(* IEC 61131-3 sources: Bachelor/LARS redcrane-simulation/plc_export/FB_InverceKinematics, 1 file *)

(* ---- RedCrane_kinematic_model.st ---- *)
(*
 *
 * File: RedCrane_kinematic_model.st
 *
 * IEC 61131-3 Structured Text (ST) code generated for subsystem "RedCrane_kinematic_model/FB_InverceKinematics"
 *
 * Model name                      : RedCrane_kinematic_model
 * Model version                   : 2.78
 * Model creator                   : sindr
 * Model last modified by          : larso
 * Model last modified on          : Mon Jan 20 08:44:51 2025
 * Model sample time               : 0.001s
 * Subsystem name                  : RedCrane_kinematic_model/FB_InverceKinematics
 * Subsystem sample time           : 0.001s
 * Simulink PLC Coder version      : 24.1 (R2024a) 19-Nov-2023
 * ST code generated on            : Mon Jan 20 09:25:34 2025
 *
 * Target IDE selection            : Beckhoff TwinCAT 3
 * Test Bench included             : No
 *
 *)
FUNCTION_BLOCK FB_InverceKinematics
VAR_INPUT
    ssMethodType: SINT;
    fXRef: LREAL;
    fYRef: LREAL;
    fZRef: LREAL;
    fXDotRef: LREAL;
    fYDotRef: LREAL;
    fZDotRef: LREAL;
    fSlewFeedback: LREAL;
    fMainFeedback: LREAL;
    fKnuckleFeedback: LREAL;
END_VAR
VAR_OUTPUT
    fSlewRef: LREAL;
    fMainRef: LREAL;
    fKnuckleRef: LREAL;
    fSlewVelRef: LREAL;
    fMainVelRef: LREAL;
    fKnuckleVelRef: LREAL;
    success: BOOL;
END_VAR
VAR
    Memory_PreviousInput: ARRAY [0..1] OF LREAL;
    Memory1_PreviousInput: LREAL;
    Memory2_PreviousInput: LREAL;
    Memory3_PreviousInput: LREAL;
    Constant4_Value: ARRAY [0..15] OF LREAL := 1.0,0.0,0.0,0.0,0.0,1.0,0.0,0.0,0.0,0.0,1.0,0.0,4.5789899999999992,
        0.3362,1.5459500000000002,1.0;
    Constant5_Value: ARRAY [0..29] OF LREAL := 0.0,0.0,1.0,0.0,0.0,0.0,0.0,-1.0,0.0,1.5685,0.0,0.25,0.0,-1.0,0.0,
        1.63847,0.0,-2.15,0.0,1.0,0.0,-1.5459500000000002,0.0,4.5789899999999992,0.0,0.0,1.0,0.3362,
        -4.5789899999999992,0.0;
    p_a: ARRAY [0..8] OF SINT := 1,0,0,0,1,0,0,0,1;
    i0_eye: eye;
    i0_pinv: pinv;
    i0_MatrixLog3: MatrixLog3;
END_VAR
VAR_TEMP
    Js: ARRAY [0..29] OF LREAL;
    T: ARRAY [0..15] OF LREAL;
    thetalist0: ARRAY [0..4] OF LREAL;
    i: DINT;
    Tsb: ARRAY [0..15] OF LREAL;
    Vs: ARRAY [0..5] OF LREAL;
    err: BOOL;
    b_i: DINT;
    c_i: DINT;
    theta: LREAL;
    d_i: DINT;
    e_i: DINT;
    b_theta: LREAL;
    se3mat: ARRAY [0..15] OF LREAL;
    omgtheta: ARRAY [0..2] OF LREAL;
    omgmat: ARRAY [0..8] OF LREAL;
    a: ARRAY [0..15] OF LREAL;
    g_a: LREAL;
    V: ARRAY [0..5] OF LREAL;
    b_R: ARRAY [0..8] OF LREAL;
    b_omgmat: ARRAY [0..8] OF LREAL;
    l_a: LREAL;
    rtb_thetaListDot: ARRAY [0..4] OF LREAL;
    d_theta: LREAL;
    g_theta: LREAL;
    thetalist0_0: LREAL;
    se3mat_0: ARRAY [0..2] OF LREAL;
    a_0: ARRAY [0..15] OF LREAL;
    tmp: ARRAY [0..8] OF LREAL;
    Tsb_0: ARRAY [0..35] OF LREAL;
    tmp_0: ARRAY [0..8] OF LREAL;
    tmp_1: ARRAY [0..29] OF LREAL;
    b_T: ARRAY [0..15] OF LREAL;
    tmp_2: ARRAY [0..8] OF LREAL;
    tmp_3: ARRAY [0..8] OF LREAL;
    tmp_4: ARRAY [0..8] OF LREAL;
    i_0: DINT;
    omgmat_tmp: DINT;
    x_tmp: LREAL;
    R_tmp: DINT;
    e_theta: LREAL;
    c_theta: LREAL;
    f_theta: LREAL;
    h_theta: LREAL;
    i_theta: LREAL;
    j_theta: LREAL;
END_VAR
CASE ssMethodType OF
    SS_INITIALIZE:
        (* SystemInitialize for Atomic SubSystem: '<Root>/FB_InverceKinematics' *)
        (* InitializeConditions for Memory: '<S1>/Memory' *)
        Memory_PreviousInput[0] := 0.0;
        Memory_PreviousInput[1] := 0.0;
        (* InitializeConditions for Memory: '<S1>/Memory1' *)
        Memory1_PreviousInput := -0.39269908169872414;
        (* InitializeConditions for Memory: '<S1>/Memory2' *)
        Memory2_PreviousInput := 0.0;
        (* InitializeConditions for Memory: '<S1>/Memory3' *)
        Memory3_PreviousInput := 0.0;
        (* End of SystemInitialize for SubSystem: '<Root>/FB_InverceKinematics' *)
    SS_STEP:
        (* Outputs for Atomic SubSystem: '<Root>/FB_InverceKinematics' *)
        (* MATLAB Function: '<S1>/inverceKinematics' incorporates:
         *  Memory: '<S1>/Memory'
         *  Memory: '<S1>/Memory1'
         *  Memory: '<S1>/Memory2'
         *  Memory: '<S1>/Memory3' *)
        thetalist0[0] := Memory3_PreviousInput;
        thetalist0[1] := Memory2_PreviousInput;
        thetalist0[2] := Memory1_PreviousInput;
        thetalist0[3] := Memory_PreviousInput[0];
        thetalist0[4] := Memory_PreviousInput[1];
        (* End of Outputs for SubSystem: '<Root>/FB_InverceKinematics' *)
        (* MATLAB Function 'FB_InverceKinematics/inverceKinematics': '<S2>:1' *)
        (* '<S2>:1:4' if(t <= Ts*1.1) *)
        (* Explicitly pre-assign outputs *)
        (* '<S2>:1:9' thetaList    = zeros(5,1); *)
        (* '<S2>:1:10' thetaListDot = zeros(5,1); *)
        (* '<S2>:1:11' success      = false; *)
        (* or 0 if you prefer numeric *)
        (* '<S2>:1:14' T = [1 0 0 x; *)
        (* '<S2>:1:15'     0 1 0 y; *)
        (* '<S2>:1:16'     0 0 1 z; *)
        (* '<S2>:1:17'     0 0 0 1]; *)
        (* Outputs for Atomic SubSystem: '<Root>/FB_InverceKinematics' *)
        (* MATLAB Function: '<S1>/inverceKinematics' *)
        T[0] := 1.0;
        T[4] := 0.0;
        T[8] := 0.0;
        T[12] := fXRef;
        T[1] := 0.0;
        T[5] := 1.0;
        T[9] := 0.0;
        T[13] := fYRef;
        T[2] := 0.0;
        T[6] := 0.0;
        T[10] := 1.0;
        T[14] := fZRef;
        T[3] := 0.0;
        T[7] := 0.0;
        T[11] := 0.0;
        T[15] := 1.0;
        (* '<S2>:1:20' [thetaOut, successOut] = IKinSpace(SList, M, T, thetaList0, 0.00001, 0.0000001); *)
        (* *** CHAPTER 6: INVERSE KINEMATICS *** *)
        (* Takes Slist: The joint screw axes in the space frame when the manipulator *)
        (* is at the home position, in the format of a matrix with the *)
        (* screw axes as the columns, *)
        (* M: The home configuration of the end-effector, *)
        (* T: The desired end-effector configuration Tsd, *)
        (* thetalist0: An initial guess of joint angles that are close to  *)
        (* satisfying Tsd, *)
        (* eomg: A small positive tolerance on the end-effector orientation  *)
        (* error. The returned joint angles must give an end-effector  *)
        (* orientation error less than eomg, *)
        (* ev: A small positive tolerance on the end-effector linear position  *)
        (* error. The returned joint angles must give an end-effector  *)
        (* position error less than ev. *)
        (* Returns thetalist: Joint angles that achieve T within the specified  *)
        (* tolerances, *)
        (* success: A logical value where TRUE means that the function found *)
        (* a solution and FALSE means that it ran through the set  *)
        (* number of maximum iterations without finding a solution *)
        (* within the tolerances eomg and ev. *)
        (* Uses an iterative Newton-Raphson root-finding method. *)
        (* The maximum number of iterations before the algorithm is terminated has  *)
        (* been hardcoded in as a variable called maxiterations. It is set to 20 at  *)
        (* the start of the function, but can be changed if needed.   *)
        (* Example Inputs: *)

        (* clear; clc; *)
        (* Slist = [[0; 0;  1;  4; 0;    0], ... *)
        (* [0; 0;  0;  0; 1;    0], ... *)
        (* [0; 0; -1; -6; 0; -0.1]]; *)
        (* M = [[-1, 0, 0, 0]; [0, 1, 0, 6]; [0, 0, -1, 2]; [0, 0, 0, 1]]; *)
        (* T = [[0, 1, 0, -5]; [1, 0, 0, 4]; [0, 0, -1, 1.6858]; [0, 0, 0, 1]]; *)
        (* thetalist0 = [1.5; 2.5; 3]; *)
        (* eomg = 0.01; *)
        (* ev = 0.001; *)
        (* [thetalist, success] = IKinSpace(Slist, M, T, thetalist0, eomg, ev) *)

        (* Output: *)
        (* thetalist = *)
        (* 1.5707 *)
        (* 2.9997 *)
        (* 3.1415 *)
        (* success = *)
        (* 1 *)
        (* 'IKinSpace:48' thetalist = thetalist0; *)
        (* 'IKinSpace:49' i = 0; *)
        i := 0;
        (* End of Outputs for SubSystem: '<Root>/FB_InverceKinematics' *)
        (* 'IKinSpace:50' maxiterations = 20; *)
        (* 'IKinSpace:51' Tsb = FKinSpace(M, Slist, thetalist); *)
        (* Outputs for Atomic SubSystem: '<Root>/FB_InverceKinematics' *)
        (* MATLAB Function: '<S1>/inverceKinematics' incorporates:
         *  Constant: '<S1>/Constant4' *)
        FOR i_0 := 0 TO 15 DO
            Tsb[i_0] := Constant4_Value[i_0];
        END_FOR;
        (* End of Outputs for SubSystem: '<Root>/FB_InverceKinematics' *)
        (* *** CHAPTER 4: FORWARD KINEMATICS *** *)
        (* Takes M: the home configuration (position and orientation) of the  *)
        (* end-effector, *)
        (* Slist: The joint screw axes in the space frame when the manipulator *)
        (* is at the home position, *)
        (* thetalist: A list of joint coordinates. *)
        (* Returns T in SE(3) representing the end-effector frame, when the joints  *)
        (* are at the specified coordinates (i.t.o Space Frame). *)
        (* Example Inputs: *)

        (* clear; clc; *)
        (* M = [[-1, 0, 0, 0]; [0, 1, 0, 6]; [0, 0, -1, 2]; [0, 0, 0, 1]]; *)
        (* Slist = [[0; 0;  1;  4; 0;    0], ... *)
        (* [0; 0;  0;  0; 1;    0], ... *)
        (* [0; 0; -1; -6; 0; -0.1]]; *)
        (* thetalist =[pi / 2; 3; pi]; *)
        (* T = FKinSpace(M, Slist, thetalist) *)

        (* Output: *)
        (* T = *)
        (* -0.0000    1.0000         0   -5.0000 *)
        (* 1.0000    0.0000         0    4.0000 *)
        (* 0         0   -1.0000    1.6858 *)
        (* 0         0         0    1.0000 *)
        (* 'FKinSpace:27' T = M; *)
        (* 'FKinSpace:28' for i = size(thetalist, 1): -1: 1 *)
        (* Outputs for Atomic SubSystem: '<Root>/FB_InverceKinematics' *)
        (* MATLAB Function: '<S1>/inverceKinematics' *)
        se3mat[0] := 0.0;
        se3mat[5] := 0.0;
        se3mat[10] := 0.0;
        se3mat[3] := 0.0;
        se3mat[7] := 0.0;
        se3mat[11] := 0.0;
        se3mat[15] := 0.0;
        (* End of Outputs for SubSystem: '<Root>/FB_InverceKinematics' *)
        (* Outputs for Atomic SubSystem: '<Root>/FB_InverceKinematics' *)
        (* MATLAB Function: '<S1>/inverceKinematics' *)
        (* End of Outputs for SubSystem: '<Root>/FB_InverceKinematics' *)
        (* Outputs for Atomic SubSystem: '<Root>/FB_InverceKinematics' *)
        (* MATLAB Function: '<S1>/inverceKinematics' incorporates:
         *  Constant: '<S1>/Constant5' *)
        FOR c_i := 0 TO 4 DO
            (* 'FKinSpace:29' T = MatrixExp6(VecTose3(Slist(:, i) * thetalist(i))) * T; *)
            thetalist0_0 := thetalist0[4 - c_i];
            FOR i_0 := 0 TO 5 DO
                V[i_0] := Constant5_Value[((4 - c_i) * 6) + i_0] * thetalist0_0;
            END_FOR;
            (* *** CHAPTER 3: RIGID-BODY MOTIONS *** *)
            (* Takes a 6-vector (representing a spatial velocity). *)
            (* Returns the corresponding 4x4 se(3) matrix. *)
            (* Example Input: *)

            (* clear; clc; *)
            (* V = [1; 2; 3; 4; 5; 6]; *)
            (* se3mat = VecTose3(V) *)

            (* Output: *)
            (* se3mat = *)
            (* 0    -3     2     4 *)
            (* 3     0    -1     5 *)
            (* -2     1     0     6 *)
            (* 0     0     0     0  *)
            (* 'VecTose3:18' se3mat = [VecToso3(V(1: 3)), V(4: 6); 0, 0, 0, 0]; *)
            (* *** CHAPTER 3: RIGID-BODY MOTIONS *** *)
            (* Takes a 3-vector (angular velocity). *)
            (* Returns the skew symmetric matrix in so(3). *)
            (* Example Input: *)

            (* clear; clc; *)
            (* omg = [1; 2; 3]; *)
            (* so3mat = VecToso3(omg) *)

            (* Output: *)
            (* so3mat = *)
            (* 0    -3     2 *)
            (* 3     0    -1 *)
            (* -2     1     0 *)
            (* 'VecToso3:17' so3mat = [0, -omg(3), omg(2); omg(3), 0, -omg(1); -omg(2), omg(1), 0]; *)
            se3mat[4] :=  -V[2];
            se3mat[8] := V[1];
            se3mat[1] := V[2];
            se3mat[9] :=  -V[0];
            se3mat[2] :=  -V[1];
            se3mat[6] := V[0];
            se3mat[12] := V[3];
            se3mat[13] := V[4];
            se3mat[14] := V[5];
            (* *** CHAPTER 3: RIGID-BODY MOTIONS *** *)
            (* Takes a se(3) representation of exponential coordinates. *)
            (* Returns a T matrix in SE(3) that is achieved by traveling along/about the  *)
            (* screw axis S for a distance theta from an initial configuration T = I. *)
            (* Example Input: *)

            (* clear; clc; *)
            (* se3mat = [ 0,      0,       0,      0; *)
            (* 0,      0, -1.5708, 2.3562; *)
            (* 0, 1.5708,       0, 2.3562; *)
            (* 0,      0,       0,      0] *)
            (* T = MatrixExp6(se3mat) *)

            (* Output: *)
            (* T = *)
            (* 1.0000         0         0         0 *)
            (* 0    0.0000   -1.0000   -0.0000 *)
            (* 0    1.0000    0.0000    3.0000 *)
            (* 0         0         0    1.0000  *)
            (* 'MatrixExp6:22' omgtheta = so3ToVec(se3mat(1: 3, 1: 3)); *)
            (* *** CHAPTER 3: RIGID-BODY MOTIONS *** *)
            (* Takes a 3x3 skew-symmetric matrix (an element of so(3)). *)
            (* Returns the corresponding 3-vector (angular velocity). *)
            (* Example Input:  *)

            (* clear; clc; *)
            (* so3mat = [[0, -3, 2]; [3, 0, -1]; [-2, 1, 0]]; *)
            (* omg = so3ToVec(so3mat)   *)

            (* Output: *)
            (* omg = *)
            (* 1 *)
            (* 2 *)
            (* 3 *)
            (* 'so3ToVec:17' omg = [so3mat(3, 2); so3mat(1, 3); so3mat(2, 1)]; *)
            (* 'MatrixExp6:23' if NearZero(norm(omgtheta)) *)
            (* *** BASIC HELPER FUNCTIONS *** *)
            (* Takes a scalar. *)
            (* Checks if the scalar is small enough to be neglected. *)
            (* Example Input: *)

            (* clear; clc; *)
            (* near = -1e-7; *)
            (* judge = NearZero(near) *)

            (* Output: *)
            (* judge = *)
            (* 1 *)
            (* 'NearZero:15' judge = norm(near) < 1e-6; *)
            se3mat_0[0] := V[0];
            se3mat_0[1] := V[1];
            se3mat_0[2] := V[2];
            d_theta := norm(x := se3mat_0);
            IF ABS(d_theta) < 1.0E-6 THEN
                (* 'MatrixExp6:24' T = [eye(3), se3mat(1: 3, 4); 0, 0, 0, 1]; *)
                i0_eye();
                tmp_0 := i0_eye.I;
                FOR i_0 := 0 TO 2 DO
                    R_tmp := DWORD_TO_DINT(SHL(DINT_TO_DWORD(i_0), 2));
                    a[R_tmp] := tmp_0[3 * i_0];
                    a[R_tmp + 1] := tmp_0[(3 * i_0) + 1];
                    a[R_tmp + 2] := tmp_0[(3 * i_0) + 2];
                    a[i_0 + 12] := se3mat[i_0 + 12];
                END_FOR;
                a[3] := 0.0;
                a[7] := 0.0;
                a[11] := 0.0;
                a[15] := 1.0;
            ELSE
                (* 'MatrixExp6:25' else *)
                (* 'MatrixExp6:26' [omghat, theta] = AxisAng3(omgtheta); *)
                (* *** CHAPTER 3: RIGID-BODY MOTIONS *** *)
                (* Takes A 3-vector of exponential coordinates for rotation. *)
                (* Returns the unit rotation axis omghat and the corresponding rotation  *)
                (* angle theta. *)
                (* Example Input: *)

                (* clear; clc; *)
                (* expc3 = [1; 2; 3]; *)
                (* [omghat, theta] = AxisAng3(expc3)   *)

                (* Output: *)
                (* omghat = *)
                (* 0.2673 *)
                (* 0.5345 *)
                (* 0.8018 *)
                (* theta = *)
                (* 3.7417 *)
                (* 'AxisAng3:20' theta = norm(expc3); *)
                (* 'AxisAng3:21' omghat = expc3 / theta; *)
                (* 'MatrixExp6:27' omgmat = se3mat(1: 3, 1: 3) / theta; *)
                FOR i_0 := 0 TO 2 DO
                    omgmat_tmp := DWORD_TO_DINT(SHL(DINT_TO_DWORD(i_0), 2));
                    omgmat[3 * i_0] := se3mat[omgmat_tmp] / d_theta;
                    omgmat[(3 * i_0) + 1] := se3mat[omgmat_tmp + 1] / d_theta;
                    omgmat[(3 * i_0) + 2] := se3mat[omgmat_tmp + 2] / d_theta;
                END_FOR;
                (* 'MatrixExp6:28' T = [MatrixExp3(se3mat(1: 3, 1: 3)), ... *)
                (* 'MatrixExp6:29'          (eye(3) * theta + (1 - cos(theta)) * omgmat ... *)
                (* 'MatrixExp6:30'           + (theta - sin(theta)) * omgmat * omgmat) ... *)
                (* 'MatrixExp6:31'             * se3mat(1: 3, 4) / theta; *)
                (* 'MatrixExp6:32'          0, 0, 0, 1]; *)
                thetalist0_0 := 1.0 - COS(d_theta);
                g_a := d_theta - SIN(d_theta);
                (* *** CHAPTER 3: RIGID-BODY MOTIONS *** *)
                (* Takes a 3x3 so(3) representation of exponential coordinates. *)
                (* Returns R in SO(3) that is achieved by rotating about omghat by theta  *)
                (* from an initial orientation R = I. *)
                (* Example Input: *)

                (* clear; clc; *)
                (* so3mat = [[0, -3, 2]; [3, 0, -1]; [-2, 1, 0]]; *)
                (* R = MatrixExp3(so3mat)   *)

                (* Output: *)
                (* R = *)
                (* -0.6949    0.7135    0.0893 *)
                (* -0.1920   -0.3038    0.9332 *)
                (* 0.6930    0.6313    0.3481 *)
                (* 'MatrixExp3:18' omgtheta = so3ToVec(so3mat); *)
                (* *** CHAPTER 3: RIGID-BODY MOTIONS *** *)
                (* Takes a 3x3 skew-symmetric matrix (an element of so(3)). *)
                (* Returns the corresponding 3-vector (angular velocity). *)
                (* Example Input:  *)

                (* clear; clc; *)
                (* so3mat = [[0, -3, 2]; [3, 0, -1]; [-2, 1, 0]]; *)
                (* omg = so3ToVec(so3mat)   *)

                (* Output: *)
                (* omg = *)
                (* 1 *)
                (* 2 *)
                (* 3 *)
                (* 'so3ToVec:17' omg = [so3mat(3, 2); so3mat(1, 3); so3mat(2, 1)]; *)
                (* 'MatrixExp3:19' if NearZero(norm(omgtheta)) *)
                (* *** BASIC HELPER FUNCTIONS *** *)
                (* Takes a scalar. *)
                (* Checks if the scalar is small enough to be neglected. *)
                (* Example Input: *)

                (* clear; clc; *)
                (* near = -1e-7; *)
                (* judge = NearZero(near) *)

                (* Output: *)
                (* judge = *)
                (* 1 *)
                (* 'NearZero:15' judge = norm(near) < 1e-6; *)
                se3mat_0[0] := V[0];
                se3mat_0[1] := V[1];
                se3mat_0[2] := V[2];
                g_theta := norm(x := se3mat_0);
                IF ABS(g_theta) < 1.0E-6 THEN
                    (* 'MatrixExp3:20' R = eye(3); *)
                    i0_eye();
                    b_R := i0_eye.I;
                ELSE
                    (* 'MatrixExp3:21' else *)
                    (* 'MatrixExp3:22' [omghat, theta] = AxisAng3(omgtheta); *)
                    (* *** CHAPTER 3: RIGID-BODY MOTIONS *** *)
                    (* Takes A 3-vector of exponential coordinates for rotation. *)
                    (* Returns the unit rotation axis omghat and the corresponding rotation  *)
                    (* angle theta. *)
                    (* Example Input: *)

                    (* clear; clc; *)
                    (* expc3 = [1; 2; 3]; *)
                    (* [omghat, theta] = AxisAng3(expc3)   *)

                    (* Output: *)
                    (* omghat = *)
                    (* 0.2673 *)
                    (* 0.5345 *)
                    (* 0.8018 *)
                    (* theta = *)
                    (* 3.7417 *)
                    (* 'AxisAng3:20' theta = norm(expc3); *)
                    (* 'AxisAng3:21' omghat = expc3 / theta; *)
                    (* 'MatrixExp3:23' omgmat = so3mat / theta; *)
                    FOR i_0 := 0 TO 2 DO
                        omgmat_tmp := DWORD_TO_DINT(SHL(DINT_TO_DWORD(i_0), 2));
                        b_omgmat[3 * i_0] := se3mat[omgmat_tmp] / g_theta;
                        b_omgmat[(3 * i_0) + 1] := se3mat[omgmat_tmp + 1] / g_theta;
                        b_omgmat[(3 * i_0) + 2] := se3mat[omgmat_tmp + 2] / g_theta;
                    END_FOR;
                    (* 'MatrixExp3:24' R = eye(3) + sin(theta) * omgmat + (1 - cos(theta)) * omgmat * omgmat; *)
                    l_a := SIN(g_theta);
                    x_tmp := COS(g_theta);
                    i0_eye();
                    tmp_0 := i0_eye.I;
                    FOR i_0 := 0 TO 2 DO
                        FOR omgmat_tmp := 0 TO 2 DO
                            R_tmp := (3 * omgmat_tmp) + i_0;
                            b_R[R_tmp] := (((((1.0 - x_tmp) * b_omgmat[i_0 + 3]) * b_omgmat[(3 * omgmat_tmp) + 1]) + (((1.0 - x_tmp) * b_omgmat[i_0]) * b_omgmat[3 * omgmat_tmp])) + ((b_omgmat[i_0 + 6] * (1.0 - x_tmp)) * b_omgmat[(3 * omgmat_tmp) + 2])) + ((b_omgmat[R_tmp] * l_a) + tmp_0[R_tmp]);
                        END_FOR;
                    END_FOR;
                END_IF;
                FOR i_0 := 0 TO 2 DO
                    x_tmp := 0.0;
                    FOR omgmat_tmp := 0 TO 2 DO
                        R_tmp := (3 * omgmat_tmp) + i_0;
                        x_tmp := ((((((omgmat[i_0 + 3] * g_a) * omgmat[(3 * omgmat_tmp) + 1]) + ((g_a * omgmat[i_0]) * omgmat[3 * omgmat_tmp])) + ((omgmat[i_0 + 6] * g_a) * omgmat[(3 * omgmat_tmp) + 2])) + ((SINT_TO_LREAL(p_a[R_tmp]) * d_theta) + (omgmat[R_tmp] * thetalist0_0))) * se3mat[omgmat_tmp + 12]) + x_tmp;
                        a[omgmat_tmp + (i_0 * 4)] := b_R[(3 * i_0) + omgmat_tmp];
                    END_FOR;
                    a[i_0 + 12] := x_tmp / d_theta;
                END_FOR;
                a[3] := 0.0;
                a[7] := 0.0;
                a[11] := 0.0;
                a[15] := 1.0;
            END_IF;
            FOR i_0 := 0 TO 3 DO
                thetalist0_0 := a[i_0 + 4];
                g_a := a[i_0];
                l_a := a[i_0 + 8];
                x_tmp := a[i_0 + 12];
                FOR omgmat_tmp := 0 TO 3 DO
                    R_tmp := DWORD_TO_DINT(SHL(DINT_TO_DWORD(omgmat_tmp), 2));
                    a_0[i_0 + R_tmp] := (((Tsb[R_tmp + 1] * thetalist0_0) + (Tsb[R_tmp] * g_a)) + (Tsb[R_tmp + 2] * l_a)) + (Tsb[R_tmp + 3] * x_tmp);
                END_FOR;
            END_FOR;
            FOR i_0 := 0 TO 15 DO
                Tsb[i_0] := a_0[i_0];
            END_FOR;
        END_FOR;
        (* End of Outputs for SubSystem: '<Root>/FB_InverceKinematics' *)
        (* 'IKinSpace:52' Vs = Adjoint(Tsb) * se3ToVec(MatrixLog6(TransInv(Tsb) * T)); *)
        (* *** CHAPTER 3: RIGID-BODY MOTIONS *** *)
        (* Takes a transformation matrix T. *)
        (* Returns its inverse.  *)
        (* Uses the structure of transformation matrices to avoid taking a matrix *)
        (* inverse, for efficiency. *)
        (* Example Input: *)

        (* clear; clc; *)
        (* T = [[1, 0, 0, 0]; [0, 0, -1, 0]; [0, 1, 0, 3]; [0, 0, 0, 1]]; *)
        (* invT = TransInv(T) *)

        (* Ouput: *)
        (* invT = *)
        (* 1     0     0     0 *)
        (* 0     0     1    -3 *)
        (* 0    -1     0     0 *)
        (* 0     0     0     1 *)
        (* 'TransInv:20' [R, p] = TransToRp(T); *)
        (* *** CHAPTER 3: RIGID-BODY MOTIONS *** *)
        (* Takes the transformation matrix T in SE(3)  *)
        (* Returns R: the corresponding rotation matrix *)
        (* p: the corresponding position vector . *)
        (* Example Input: *)

        (* clear; clc; *)
        (* T = [[1, 0, 0, 0]; [0, 0, -1, 0]; [0, 1, 0, 3]; [0, 0, 0, 1]]; *)
        (* [R, p] = TransToRp(T) *)

        (* Output: *)
        (* R = *)
        (* 1     0     0 *)
        (* 0     0    -1 *)
        (* 0     1     0 *)
        (* p = *)
        (* 0 *)
        (* 0 *)
        (* 3 *)
        (* 'TransToRp:22' R = T(1: 3, 1: 3); *)
        (* 'TransToRp:23' p = T(1: 3, 4); *)
        (* 'TransInv:21' invT = [transpose(R), -transpose(R) * p; 0, 0, 0, 1]; *)
        (* Outputs for Atomic SubSystem: '<Root>/FB_InverceKinematics' *)
        (* MATLAB Function: '<S1>/inverceKinematics' *)
        FOR i_0 := 0 TO 2 DO
            omgmat[3 * i_0] := Tsb[i_0];
            omgmat[(3 * i_0) + 1] := Tsb[i_0 + 4];
            omgmat[(3 * i_0) + 2] := Tsb[i_0 + 8];
        END_FOR;
        (* End of Outputs for SubSystem: '<Root>/FB_InverceKinematics' *)
        (* Outputs for Atomic SubSystem: '<Root>/FB_InverceKinematics' *)
        (* MATLAB Function: '<S1>/inverceKinematics' *)
        FOR i_0 := 0 TO 8 DO
            b_R[i_0] :=  -omgmat[i_0];
        END_FOR;
        (* End of Outputs for SubSystem: '<Root>/FB_InverceKinematics' *)
        (* Outputs for Atomic SubSystem: '<Root>/FB_InverceKinematics' *)
        (* MATLAB Function: '<S1>/inverceKinematics' *)
        thetalist0_0 := Tsb[13];
        g_a := Tsb[12];
        l_a := Tsb[14];
        FOR i_0 := 0 TO 2 DO
            omgmat_tmp := DWORD_TO_DINT(SHL(DINT_TO_DWORD(i_0), 2));
            se3mat[omgmat_tmp] := omgmat[3 * i_0];
            se3mat[omgmat_tmp + 1] := omgmat[(3 * i_0) + 1];
            se3mat[omgmat_tmp + 2] := omgmat[(3 * i_0) + 2];
            se3mat[i_0 + 12] := ((b_R[i_0 + 3] * thetalist0_0) + (b_R[i_0] * g_a)) + (b_R[i_0 + 6] * l_a);
        END_FOR;
        se3mat[3] := 0.0;
        se3mat[7] := 0.0;
        se3mat[11] := 0.0;
        se3mat[15] := 1.0;
        (* End of Outputs for SubSystem: '<Root>/FB_InverceKinematics' *)
        (* Outputs for Atomic SubSystem: '<Root>/FB_InverceKinematics' *)
        (* MATLAB Function: '<S1>/inverceKinematics' *)
        FOR i_0 := 0 TO 3 DO
            R_tmp := DWORD_TO_DINT(SHL(DINT_TO_DWORD(i_0), 2));
            thetalist0_0 := T[R_tmp + 1];
            g_a := T[R_tmp];
            l_a := T[R_tmp + 2];
            x_tmp := T[R_tmp + 3];
            FOR omgmat_tmp := 0 TO 3 DO
                a_0[omgmat_tmp + R_tmp] := (((thetalist0_0 * se3mat[omgmat_tmp + 4]) + (g_a * se3mat[omgmat_tmp])) + (l_a * se3mat[omgmat_tmp + 8])) + (x_tmp * se3mat[omgmat_tmp + 12]);
            END_FOR;
        END_FOR;
        (* End of Outputs for SubSystem: '<Root>/FB_InverceKinematics' *)
        (* *** CHAPTER 3: RIGID-BODY MOTIONS *** *)
        (* Takes a transformation matrix T in SE(3). *)
        (* Returns the corresponding se(3) representation of exponential  *)
        (* coordinates. *)
        (* Example Input: *)

        (* clear; clc; *)
        (* T = [[1, 0, 0, 0]; [0, 0, -1, 0]; [0, 1, 0, 3]; [0, 0, 0, 1]]; *)
        (* expmat = MatrixLog6(T) *)

        (* Output: *)
        (* expc6 = *)
        (* 0         0         0         0 *)
        (* 0         0   -1.5708    2.3562 *)
        (* 0    1.5708         0    2.3562 *)
        (* 0         0         0         0 *)
        (* 'MatrixLog6:19' [R, p] = TransToRp(T); *)
        (* *** CHAPTER 3: RIGID-BODY MOTIONS *** *)
        (* Takes the transformation matrix T in SE(3)  *)
        (* Returns R: the corresponding rotation matrix *)
        (* p: the corresponding position vector . *)
        (* Example Input: *)

        (* clear; clc; *)
        (* T = [[1, 0, 0, 0]; [0, 0, -1, 0]; [0, 1, 0, 3]; [0, 0, 0, 1]]; *)
        (* [R, p] = TransToRp(T) *)

        (* Output: *)
        (* R = *)
        (* 1     0     0 *)
        (* 0     0    -1 *)
        (* 0     1     0 *)
        (* p = *)
        (* 0 *)
        (* 0 *)
        (* 3 *)
        (* 'TransToRp:22' R = T(1: 3, 1: 3); *)
        (* 'TransToRp:23' p = T(1: 3, 4); *)
        (* 'MatrixLog6:20' omgmat = MatrixLog3(R); *)
        (* Outputs for Atomic SubSystem: '<Root>/FB_InverceKinematics' *)
        (* MATLAB Function: '<S1>/inverceKinematics' *)
        FOR i_0 := 0 TO 2 DO
            R_tmp := DWORD_TO_DINT(SHL(DINT_TO_DWORD(i_0), 2));
            b_R[3 * i_0] := a_0[R_tmp];
            b_R[(3 * i_0) + 1] := a_0[R_tmp + 1];
            b_R[(3 * i_0) + 2] := a_0[R_tmp + 2];
        END_FOR;
        i0_MatrixLog3(b_R := b_R);
        omgmat := i0_MatrixLog3.so3mat;
        (* End of Outputs for SubSystem: '<Root>/FB_InverceKinematics' *)
        (* 'MatrixLog6:21' if isequal(omgmat, zeros(3)) *)
        (* Outputs for Atomic SubSystem: '<Root>/FB_InverceKinematics' *)
        (* MATLAB Function: '<S1>/inverceKinematics' *)
        FOR i_0 := 0 TO 8 DO
            tmp_0[i_0] := 0.0;
        END_FOR;
        IF isequal(varargin_1 := omgmat, varargin_2 := tmp_0) THEN
            (* 'MatrixLog6:22' expmat = [zeros(3), T(1: 3, 4); 0, 0, 0, 0]; *)
            FOR i_0 := 0 TO 2 DO
                omgmat_tmp := DWORD_TO_DINT(SHL(DINT_TO_DWORD(i_0), 2));
                se3mat[omgmat_tmp] := 0.0;
                se3mat[omgmat_tmp + 1] := 0.0;
                se3mat[omgmat_tmp + 2] := 0.0;
                se3mat[i_0 + 12] := a_0[i_0 + 12];
            END_FOR;
            se3mat[3] := 0.0;
            se3mat[7] := 0.0;
            se3mat[11] := 0.0;
            se3mat[15] := 0.0;
        ELSE
            (* 'MatrixLog6:23' else *)
            (* 'MatrixLog6:24' theta = acos((trace(R) - 1) / 2); *)
            theta := ACOS((((a_0[0] + a_0[5]) + a_0[10]) - 1.0) / 2.0);
            (* 'MatrixLog6:25' expmat = [omgmat, (eye(3) - omgmat / 2 ... *)
            (* 'MatrixLog6:26'                       + (1 / theta - cot(theta / 2) / 2) ... *)
            (* 'MatrixLog6:27'                         * omgmat * omgmat / theta) * p; *)
            (* 'MatrixLog6:28'               0, 0, 0, 0]; *)
            thetalist0_0 := (1.0 / theta) - ((1.0 / TAN(theta / 2.0)) / 2.0);
            i0_eye();
            tmp_0 := i0_eye.I;
            FOR i_0 := 0 TO 2 DO
                x_tmp := 0.0;
                FOR omgmat_tmp := 0 TO 2 DO
                    R_tmp := (3 * omgmat_tmp) + i_0;
                    x_tmp := (((((((omgmat[i_0 + 3] * thetalist0_0) * omgmat[(3 * omgmat_tmp) + 1]) + ((thetalist0_0 * omgmat[i_0]) * omgmat[3 * omgmat_tmp])) + ((omgmat[i_0 + 6] * thetalist0_0) * omgmat[(3 * omgmat_tmp) + 2])) / theta) + (tmp_0[R_tmp] - (omgmat[R_tmp] / 2.0))) * a_0[omgmat_tmp + 12]) + x_tmp;
                    se3mat[omgmat_tmp + (i_0 * 4)] := omgmat[(3 * i_0) + omgmat_tmp];
                END_FOR;
                se3mat[i_0 + 12] := x_tmp;
            END_FOR;
            se3mat[3] := 0.0;
            se3mat[7] := 0.0;
            se3mat[11] := 0.0;
            se3mat[15] := 0.0;
        END_IF;
        (* End of Outputs for SubSystem: '<Root>/FB_InverceKinematics' *)
        (* *** CHAPTER 3: RIGID-BODY MOTIONS *** *)
        (* Takes T a transformation matrix SE3.  *)
        (* Returns the corresponding 6x6 adjoint representation [AdT]. *)
        (* Example Input: *)

        (* clear; clc; *)
        (* T = [[1, 0, 0, 0]; [0, 0, -1, 0]; [0, 1, 0, 3]; [0, 0, 0, 1]]; *)
        (* AdT = Adjoint(T) *)

        (* Output: *)
        (* AdT = *)
        (* 1     0     0     0     0     0 *)
        (* 0     0    -1     0     0     0 *)
        (* 0     1     0     0     0     0 *)
        (* 0     0     3     1     0     0 *)
        (* 3     0     0     0     0    -1 *)
        (* 0     0     0     0     1     0 *)
        (* 'Adjoint:20' [R, p] = TransToRp(T); *)
        (* *** CHAPTER 3: RIGID-BODY MOTIONS *** *)
        (* Takes the transformation matrix T in SE(3)  *)
        (* Returns R: the corresponding rotation matrix *)
        (* p: the corresponding position vector . *)
        (* Example Input: *)

        (* clear; clc; *)
        (* T = [[1, 0, 0, 0]; [0, 0, -1, 0]; [0, 1, 0, 3]; [0, 0, 0, 1]]; *)
        (* [R, p] = TransToRp(T) *)

        (* Output: *)
        (* R = *)
        (* 1     0     0 *)
        (* 0     0    -1 *)
        (* 0     1     0 *)
        (* p = *)
        (* 0 *)
        (* 0 *)
        (* 3 *)
        (* 'TransToRp:22' R = T(1: 3, 1: 3); *)
        (* 'TransToRp:23' p = T(1: 3, 4); *)
        (* 'Adjoint:21' AdT = [R, zeros(3); VecToso3(p) * R, R]; *)
        (* *** CHAPTER 3: RIGID-BODY MOTIONS *** *)
        (* Takes a 3-vector (angular velocity). *)
        (* Returns the skew symmetric matrix in so(3). *)
        (* Example Input: *)

        (* clear; clc; *)
        (* omg = [1; 2; 3]; *)
        (* so3mat = VecToso3(omg) *)

        (* Output: *)
        (* so3mat = *)
        (* 0    -3     2 *)
        (* 3     0    -1 *)
        (* -2     1     0 *)
        (* 'VecToso3:17' so3mat = [0, -omg(3), omg(2); omg(3), 0, -omg(1); -omg(2), omg(1), 0]; *)
        (* *** CHAPTER 3: RIGID-BODY MOTIONS *** *)
        (* Takes se3mat a 4x4 se(3) matrix *)
        (* Returns the corresponding 6-vector (representing spatial velocity). *)
        (* Example Input: *)

        (* clear; clc; *)
        (* se3mat = [[0, -3, 2, 4]; [3, 0, -1, 5]; [-2, 1, 0, 6]; [0, 0, 0, 0]]; *)
        (* V = se3ToVec(se3mat) *)

        (* Output: *)
        (* V = *)
        (* 1 *)
        (* 2 *)
        (* 3 *)
        (* 4 *)
        (* 5 *)
        (* 6 *)
        (* 'se3ToVec:20' V = [se3mat(3, 2); se3mat(1, 3); se3mat(2, 1); se3mat(1: 3, 4)]; *)
        (* Outputs for Atomic SubSystem: '<Root>/FB_InverceKinematics' *)
        (* MATLAB Function: '<S1>/inverceKinematics' *)
        tmp_0[0] := 0.0;
        tmp_0[3] :=  -Tsb[14];
        tmp_0[6] := Tsb[13];
        tmp_0[1] := Tsb[14];
        tmp_0[4] := 0.0;
        tmp_0[7] :=  -Tsb[12];
        tmp_0[2] :=  -Tsb[13];
        tmp_0[5] := Tsb[12];
        tmp_0[8] := 0.0;
        (* End of Outputs for SubSystem: '<Root>/FB_InverceKinematics' *)
        (* Outputs for Atomic SubSystem: '<Root>/FB_InverceKinematics' *)
        (* MATLAB Function: '<S1>/inverceKinematics' *)
        FOR i_0 := 0 TO 2 DO
            x_tmp := tmp_0[i_0 + 3];
            thetalist0_0 := tmp_0[i_0];
            g_a := tmp_0[i_0 + 6];
            FOR omgmat_tmp := 0 TO 2 DO
                R_tmp := DWORD_TO_DINT(SHL(DINT_TO_DWORD(omgmat_tmp), 2));
                tmp[i_0 + (3 * omgmat_tmp)] := ((Tsb[R_tmp + 1] * x_tmp) + (Tsb[R_tmp] * thetalist0_0)) + (Tsb[R_tmp + 2] * g_a);
                Tsb_0[omgmat_tmp + (6 * i_0)] := Tsb[(i_0 * 4) + omgmat_tmp];
                Tsb_0[omgmat_tmp + (6 * (i_0 + 3))] := 0.0;
            END_FOR;
        END_FOR;
        (* End of Outputs for SubSystem: '<Root>/FB_InverceKinematics' *)
        (* Outputs for Atomic SubSystem: '<Root>/FB_InverceKinematics' *)
        (* MATLAB Function: '<S1>/inverceKinematics' *)
        V[0] := se3mat[6];
        V[1] := se3mat[8];
        V[2] := se3mat[1];
        FOR i_0 := 0 TO 2 DO
            Tsb_0[(6 * i_0) + 3] := tmp[3 * i_0];
            omgmat_tmp := DWORD_TO_DINT(SHL(DINT_TO_DWORD(i_0), 2));
            R_tmp := 6 * (i_0 + 3);
            Tsb_0[R_tmp + 3] := Tsb[omgmat_tmp];
            Tsb_0[(6 * i_0) + 4] := tmp[(3 * i_0) + 1];
            Tsb_0[R_tmp + 4] := Tsb[omgmat_tmp + 1];
            Tsb_0[(6 * i_0) + 5] := tmp[(3 * i_0) + 2];
            Tsb_0[R_tmp + 5] := Tsb[omgmat_tmp + 2];
            V[i_0 + 3] := se3mat[i_0 + 12];
        END_FOR;
        (* End of Outputs for SubSystem: '<Root>/FB_InverceKinematics' *)
        (* Outputs for Atomic SubSystem: '<Root>/FB_InverceKinematics' *)
        (* MATLAB Function: '<S1>/inverceKinematics' *)
        FOR i_0 := 0 TO 5 DO
            thetalist0_0 := 0.0;
            FOR omgmat_tmp := 0 TO 5 DO
                thetalist0_0 := (Tsb_0[(6 * omgmat_tmp) + i_0] * V[omgmat_tmp]) + thetalist0_0;
            END_FOR;
            Vs[i_0] := thetalist0_0;
        END_FOR;
        (* End of Outputs for SubSystem: '<Root>/FB_InverceKinematics' *)
        (* 'IKinSpace:53' err = norm(Vs(1: 3)) > eomg || norm(Vs(4: 6)) > ev; *)
        (* Outputs for Atomic SubSystem: '<Root>/FB_InverceKinematics' *)
        (* MATLAB Function: '<S1>/inverceKinematics' incorporates:
         *  Constant: '<S1>/Constant4'
         *  Constant: '<S1>/Constant5' *)
        se3mat_0[0] := Vs[0];
        se3mat_0[1] := Vs[1];
        se3mat_0[2] := Vs[2];
        IF norm(x := se3mat_0) > 1.0E-5 THEN
            err := TRUE;
        ELSE
            se3mat_0[0] := Vs[3];
            se3mat_0[1] := Vs[4];
            se3mat_0[2] := Vs[5];
            IF norm(x := se3mat_0) > 1.0E-7 THEN
                err := TRUE;
            ELSE
                err := FALSE;
            END_IF;
        END_IF;
        (* 'IKinSpace:54' while err && i < maxiterations *)
        IF err THEN
            tmp_3[0] := 0.0;
            tmp_3[4] := 0.0;
            tmp_3[8] := 0.0;
            tmp_4[0] := 0.0;
            tmp_4[4] := 0.0;
            tmp_4[8] := 0.0;
            FOR i_0 := 0 TO 8 DO
                tmp_2[i_0] := 0.0;
            END_FOR;
        END_IF;
        WHILE err AND (i < 20) DO
            (* 'IKinSpace:55' thetalist = thetalist + pinv(JacobianSpace(Slist, thetalist)) * Vs; *)
            (* *** CHAPTER 5: VELOCITY KINEMATICS AND STATICS *** *)
            (* Takes Slist: The joint screw axes in the space frame when the manipulator *)
            (* is at the home position, in the format of a matrix with the *)
            (* screw axes as the columns, *)
            (* thetalist: A list of joint coordinates.  *)
            (* Returns the corresponding space Jacobian (6xn real numbers). *)
            (* Example Input: *)

            (* clear; clc; *)
            (* Slist = [[0; 0; 1;   0; 0.2; 0.2], ... *)
            (* [1; 0; 0;   2;   0;   3], ... *)
            (* [0; 1; 0;   0;   2;   1], ... *)
            (* [1; 0; 0; 0.2; 0.3; 0.4]]; *)
            (* thetalist = [0.2; 1.1; 0.1; 1.2]; *)
            (* Js = JacobianSpace(Slist, thetalist) *)

            (* Output: *)
            (* Js = *)
            (* 0    0.9801   -0.0901    0.9575 *)
            (* 0    0.1987    0.4446    0.2849 *)
            (* 1.0000         0    0.8912   -0.0453 *)
            (* 0    1.9522   -2.2164   -0.5116 *)
            (* 0.2000    0.4365   -2.4371    2.7754 *)
            (* 0.2000    2.9603    3.2357    2.2251 *)
            (* 'JacobianSpace:27' Js = Slist; *)
            FOR i_0 := 0 TO 29 DO
                Js[i_0] := Constant5_Value[i_0];
            END_FOR;
            (* 'JacobianSpace:28' T = eye(4); *)
            FOR i_0 := 0 TO 15 DO
                a_0[i_0] := 0.0;
            END_FOR;
            a_0[0] := 1.0;
            a_0[5] := 1.0;
            a_0[10] := 1.0;
            a_0[15] := 1.0;
            (* 'JacobianSpace:29' for i = 2: length(thetalist) *)
            se3mat[0] := 0.0;
            se3mat[5] := 0.0;
            se3mat[10] := 0.0;
            se3mat[3] := 0.0;
            se3mat[7] := 0.0;
            se3mat[11] := 0.0;
            se3mat[15] := 0.0;
            FOR d_i := 0 TO 3 DO
                (* 'JacobianSpace:30' T = T * MatrixExp6(VecTose3(Slist(:, i - 1) * thetalist(i - 1))); *)
                thetalist0_0 := thetalist0[d_i];
                FOR i_0 := 0 TO 5 DO
                    V[i_0] := Constant5_Value[(6 * d_i) + i_0] * thetalist0_0;
                END_FOR;
                (* *** CHAPTER 3: RIGID-BODY MOTIONS *** *)
                (* Takes a 6-vector (representing a spatial velocity). *)
                (* Returns the corresponding 4x4 se(3) matrix. *)
                (* Example Input: *)

                (* clear; clc; *)
                (* V = [1; 2; 3; 4; 5; 6]; *)
                (* se3mat = VecTose3(V) *)

                (* Output: *)
                (* se3mat = *)
                (* 0    -3     2     4 *)
                (* 3     0    -1     5 *)
                (* -2     1     0     6 *)
                (* 0     0     0     0  *)
                (* 'VecTose3:18' se3mat = [VecToso3(V(1: 3)), V(4: 6); 0, 0, 0, 0]; *)
                (* *** CHAPTER 3: RIGID-BODY MOTIONS *** *)
                (* Takes a 3-vector (angular velocity). *)
                (* Returns the skew symmetric matrix in so(3). *)
                (* Example Input: *)

                (* clear; clc; *)
                (* omg = [1; 2; 3]; *)
                (* so3mat = VecToso3(omg) *)

                (* Output: *)
                (* so3mat = *)
                (* 0    -3     2 *)
                (* 3     0    -1 *)
                (* -2     1     0 *)
                (* 'VecToso3:17' so3mat = [0, -omg(3), omg(2); omg(3), 0, -omg(1); -omg(2), omg(1), 0]; *)
                se3mat[4] :=  -V[2];
                se3mat[8] := V[1];
                se3mat[1] := V[2];
                se3mat[9] :=  -V[0];
                se3mat[2] :=  -V[1];
                se3mat[6] := V[0];
                se3mat[12] := V[3];
                se3mat[13] := V[4];
                se3mat[14] := V[5];
                (* *** CHAPTER 3: RIGID-BODY MOTIONS *** *)
                (* Takes a se(3) representation of exponential coordinates. *)
                (* Returns a T matrix in SE(3) that is achieved by traveling along/about the  *)
                (* screw axis S for a distance theta from an initial configuration T = I. *)
                (* Example Input: *)

                (* clear; clc; *)
                (* se3mat = [ 0,      0,       0,      0; *)
                (* 0,      0, -1.5708, 2.3562; *)
                (* 0, 1.5708,       0, 2.3562; *)
                (* 0,      0,       0,      0] *)
                (* T = MatrixExp6(se3mat) *)

                (* Output: *)
                (* T = *)
                (* 1.0000         0         0         0 *)
                (* 0    0.0000   -1.0000   -0.0000 *)
                (* 0    1.0000    0.0000    3.0000 *)
                (* 0         0         0    1.0000  *)
                (* 'MatrixExp6:22' omgtheta = so3ToVec(se3mat(1: 3, 1: 3)); *)
                (* *** CHAPTER 3: RIGID-BODY MOTIONS *** *)
                (* Takes a 3x3 skew-symmetric matrix (an element of so(3)). *)
                (* Returns the corresponding 3-vector (angular velocity). *)
                (* Example Input:  *)

                (* clear; clc; *)
                (* so3mat = [[0, -3, 2]; [3, 0, -1]; [-2, 1, 0]]; *)
                (* omg = so3ToVec(so3mat)   *)

                (* Output: *)
                (* omg = *)
                (* 1 *)
                (* 2 *)
                (* 3 *)
                (* 'so3ToVec:17' omg = [so3mat(3, 2); so3mat(1, 3); so3mat(2, 1)]; *)
                omgtheta[0] := V[0];
                omgtheta[1] := V[1];
                omgtheta[2] := V[2];
                (* 'MatrixExp6:23' if NearZero(norm(omgtheta)) *)
                (* *** BASIC HELPER FUNCTIONS *** *)
                (* Takes a scalar. *)
                (* Checks if the scalar is small enough to be neglected. *)
                (* Example Input: *)

                (* clear; clc; *)
                (* near = -1e-7; *)
                (* judge = NearZero(near) *)

                (* Output: *)
                (* judge = *)
                (* 1 *)
                (* 'NearZero:15' judge = norm(near) < 1e-6; *)
                e_theta := norm(x := omgtheta);
                IF ABS(e_theta) < 1.0E-6 THEN
                    (* 'MatrixExp6:24' T = [eye(3), se3mat(1: 3, 4); 0, 0, 0, 1]; *)
                    i0_eye();
                    tmp_0 := i0_eye.I;
                    FOR i_0 := 0 TO 2 DO
                        R_tmp := DWORD_TO_DINT(SHL(DINT_TO_DWORD(i_0), 2));
                        a[R_tmp] := tmp_0[3 * i_0];
                        a[R_tmp + 1] := tmp_0[(3 * i_0) + 1];
                        a[R_tmp + 2] := tmp_0[(3 * i_0) + 2];
                        a[i_0 + 12] := se3mat[i_0 + 12];
                    END_FOR;
                    a[3] := 0.0;
                    a[7] := 0.0;
                    a[11] := 0.0;
                    a[15] := 1.0;
                ELSE
                    (* 'MatrixExp6:25' else *)
                    (* 'MatrixExp6:26' [omghat, theta] = AxisAng3(omgtheta); *)
                    (* *** CHAPTER 3: RIGID-BODY MOTIONS *** *)
                    (* Takes A 3-vector of exponential coordinates for rotation. *)
                    (* Returns the unit rotation axis omghat and the corresponding rotation  *)
                    (* angle theta. *)
                    (* Example Input: *)

                    (* clear; clc; *)
                    (* expc3 = [1; 2; 3]; *)
                    (* [omghat, theta] = AxisAng3(expc3)   *)

                    (* Output: *)
                    (* omghat = *)
                    (* 0.2673 *)
                    (* 0.5345 *)
                    (* 0.8018 *)
                    (* theta = *)
                    (* 3.7417 *)
                    (* 'AxisAng3:20' theta = norm(expc3); *)
                    (* 'AxisAng3:21' omghat = expc3 / theta; *)
                    (* 'MatrixExp6:27' omgmat = se3mat(1: 3, 1: 3) / theta; *)
                    FOR i_0 := 0 TO 2 DO
                        omgmat_tmp := DWORD_TO_DINT(SHL(DINT_TO_DWORD(i_0), 2));
                        omgmat[3 * i_0] := se3mat[omgmat_tmp] / e_theta;
                        omgmat[(3 * i_0) + 1] := se3mat[omgmat_tmp + 1] / e_theta;
                        omgmat[(3 * i_0) + 2] := se3mat[omgmat_tmp + 2] / e_theta;
                    END_FOR;
                    (* 'MatrixExp6:28' T = [MatrixExp3(se3mat(1: 3, 1: 3)), ... *)
                    (* 'MatrixExp6:29'          (eye(3) * theta + (1 - cos(theta)) * omgmat ... *)
                    (* 'MatrixExp6:30'           + (theta - sin(theta)) * omgmat * omgmat) ... *)
                    (* 'MatrixExp6:31'             * se3mat(1: 3, 4) / theta; *)
                    (* 'MatrixExp6:32'          0, 0, 0, 1]; *)
                    thetalist0_0 := 1.0 - COS(e_theta);
                    g_a := e_theta - SIN(e_theta);
                    (* *** CHAPTER 3: RIGID-BODY MOTIONS *** *)
                    (* Takes a 3x3 so(3) representation of exponential coordinates. *)
                    (* Returns R in SO(3) that is achieved by rotating about omghat by theta  *)
                    (* from an initial orientation R = I. *)
                    (* Example Input: *)

                    (* clear; clc; *)
                    (* so3mat = [[0, -3, 2]; [3, 0, -1]; [-2, 1, 0]]; *)
                    (* R = MatrixExp3(so3mat)   *)

                    (* Output: *)
                    (* R = *)
                    (* -0.6949    0.7135    0.0893 *)
                    (* -0.1920   -0.3038    0.9332 *)
                    (* 0.6930    0.6313    0.3481 *)
                    (* 'MatrixExp3:18' omgtheta = so3ToVec(so3mat); *)
                    (* *** CHAPTER 3: RIGID-BODY MOTIONS *** *)
                    (* Takes a 3x3 skew-symmetric matrix (an element of so(3)). *)
                    (* Returns the corresponding 3-vector (angular velocity). *)
                    (* Example Input:  *)

                    (* clear; clc; *)
                    (* so3mat = [[0, -3, 2]; [3, 0, -1]; [-2, 1, 0]]; *)
                    (* omg = so3ToVec(so3mat)   *)

                    (* Output: *)
                    (* omg = *)
                    (* 1 *)
                    (* 2 *)
                    (* 3 *)
                    (* 'so3ToVec:17' omg = [so3mat(3, 2); so3mat(1, 3); so3mat(2, 1)]; *)
                    omgtheta[0] := V[0];
                    omgtheta[1] := V[1];
                    omgtheta[2] := V[2];
                    (* 'MatrixExp3:19' if NearZero(norm(omgtheta)) *)
                    (* *** BASIC HELPER FUNCTIONS *** *)
                    (* Takes a scalar. *)
                    (* Checks if the scalar is small enough to be neglected. *)
                    (* Example Input: *)

                    (* clear; clc; *)
                    (* near = -1e-7; *)
                    (* judge = NearZero(near) *)

                    (* Output: *)
                    (* judge = *)
                    (* 1 *)
                    (* 'NearZero:15' judge = norm(near) < 1e-6; *)
                    h_theta := norm(x := omgtheta);
                    IF ABS(h_theta) < 1.0E-6 THEN
                        (* 'MatrixExp3:20' R = eye(3); *)
                        i0_eye();
                        b_R := i0_eye.I;
                    ELSE
                        (* 'MatrixExp3:21' else *)
                        (* 'MatrixExp3:22' [omghat, theta] = AxisAng3(omgtheta); *)
                        (* *** CHAPTER 3: RIGID-BODY MOTIONS *** *)
                        (* Takes A 3-vector of exponential coordinates for rotation. *)
                        (* Returns the unit rotation axis omghat and the corresponding rotation  *)
                        (* angle theta. *)
                        (* Example Input: *)

                        (* clear; clc; *)
                        (* expc3 = [1; 2; 3]; *)
                        (* [omghat, theta] = AxisAng3(expc3)   *)

                        (* Output: *)
                        (* omghat = *)
                        (* 0.2673 *)
                        (* 0.5345 *)
                        (* 0.8018 *)
                        (* theta = *)
                        (* 3.7417 *)
                        (* 'AxisAng3:20' theta = norm(expc3); *)
                        (* 'AxisAng3:21' omghat = expc3 / theta; *)
                        (* 'MatrixExp3:23' omgmat = so3mat / theta; *)
                        FOR i_0 := 0 TO 2 DO
                            omgmat_tmp := DWORD_TO_DINT(SHL(DINT_TO_DWORD(i_0), 2));
                            b_omgmat[3 * i_0] := se3mat[omgmat_tmp] / h_theta;
                            b_omgmat[(3 * i_0) + 1] := se3mat[omgmat_tmp + 1] / h_theta;
                            b_omgmat[(3 * i_0) + 2] := se3mat[omgmat_tmp + 2] / h_theta;
                        END_FOR;
                        (* 'MatrixExp3:24' R = eye(3) + sin(theta) * omgmat + (1 - cos(theta)) * omgmat * omgmat; *)
                        l_a := SIN(h_theta);
                        x_tmp := COS(h_theta);
                        i0_eye();
                        tmp_0 := i0_eye.I;
                        FOR i_0 := 0 TO 2 DO
                            FOR omgmat_tmp := 0 TO 2 DO
                                R_tmp := (3 * omgmat_tmp) + i_0;
                                b_R[R_tmp] := (((((1.0 - x_tmp) * b_omgmat[i_0 + 3]) * b_omgmat[(3 * omgmat_tmp) + 1]) + (((1.0 - x_tmp) * b_omgmat[i_0]) * b_omgmat[3 * omgmat_tmp])) + ((b_omgmat[i_0 + 6] * (1.0 - x_tmp)) * b_omgmat[(3 * omgmat_tmp) + 2])) + ((b_omgmat[R_tmp] * l_a) + tmp_0[R_tmp]);
                            END_FOR;
                        END_FOR;
                    END_IF;
                    FOR i_0 := 0 TO 2 DO
                        x_tmp := 0.0;
                        FOR omgmat_tmp := 0 TO 2 DO
                            R_tmp := (3 * omgmat_tmp) + i_0;
                            x_tmp := ((((((omgmat[i_0 + 3] * g_a) * omgmat[(3 * omgmat_tmp) + 1]) + ((g_a * omgmat[i_0]) * omgmat[3 * omgmat_tmp])) + ((omgmat[i_0 + 6] * g_a) * omgmat[(3 * omgmat_tmp) + 2])) + ((SINT_TO_LREAL(p_a[R_tmp]) * e_theta) + (omgmat[R_tmp] * thetalist0_0))) * se3mat[omgmat_tmp + 12]) + x_tmp;
                            a[omgmat_tmp + (i_0 * 4)] := b_R[(3 * i_0) + omgmat_tmp];
                        END_FOR;
                        a[i_0 + 12] := x_tmp / e_theta;
                    END_FOR;
                    a[3] := 0.0;
                    a[7] := 0.0;
                    a[11] := 0.0;
                    a[15] := 1.0;
                END_IF;
                FOR i_0 := 0 TO 3 DO
                    thetalist0_0 := a_0[i_0 + 4];
                    g_a := a_0[i_0];
                    l_a := a_0[i_0 + 8];
                    x_tmp := a_0[i_0 + 12];
                    FOR omgmat_tmp := 0 TO 3 DO
                        R_tmp := DWORD_TO_DINT(SHL(DINT_TO_DWORD(omgmat_tmp), 2));
                        b_T[i_0 + R_tmp] := (((a[R_tmp + 1] * thetalist0_0) + (a[R_tmp] * g_a)) + (a[R_tmp + 2] * l_a)) + (a[R_tmp + 3] * x_tmp);
                    END_FOR;
                END_FOR;
                FOR i_0 := 0 TO 15 DO
                    a_0[i_0] := b_T[i_0];
                END_FOR;
                (* 'JacobianSpace:31' Js(:, i) = Adjoint(T) * Slist(:, i); *)
                (* *** CHAPTER 3: RIGID-BODY MOTIONS *** *)
                (* Takes T a transformation matrix SE3.  *)
                (* Returns the corresponding 6x6 adjoint representation [AdT]. *)
                (* Example Input: *)

                (* clear; clc; *)
                (* T = [[1, 0, 0, 0]; [0, 0, -1, 0]; [0, 1, 0, 3]; [0, 0, 0, 1]]; *)
                (* AdT = Adjoint(T) *)

                (* Output: *)
                (* AdT = *)
                (* 1     0     0     0     0     0 *)
                (* 0     0    -1     0     0     0 *)
                (* 0     1     0     0     0     0 *)
                (* 0     0     3     1     0     0 *)
                (* 3     0     0     0     0    -1 *)
                (* 0     0     0     0     1     0 *)
                (* 'Adjoint:20' [R, p] = TransToRp(T); *)
                (* *** CHAPTER 3: RIGID-BODY MOTIONS *** *)
                (* Takes the transformation matrix T in SE(3)  *)
                (* Returns R: the corresponding rotation matrix *)
                (* p: the corresponding position vector . *)
                (* Example Input: *)

                (* clear; clc; *)
                (* T = [[1, 0, 0, 0]; [0, 0, -1, 0]; [0, 1, 0, 3]; [0, 0, 0, 1]]; *)
                (* [R, p] = TransToRp(T) *)

                (* Output: *)
                (* R = *)
                (* 1     0     0 *)
                (* 0     0    -1 *)
                (* 0     1     0 *)
                (* p = *)
                (* 0 *)
                (* 0 *)
                (* 3 *)
                (* 'TransToRp:22' R = T(1: 3, 1: 3); *)
                (* 'TransToRp:23' p = T(1: 3, 4); *)
                (* 'Adjoint:21' AdT = [R, zeros(3); VecToso3(p) * R, R]; *)
                (* *** CHAPTER 3: RIGID-BODY MOTIONS *** *)
                (* Takes a 3-vector (angular velocity). *)
                (* Returns the skew symmetric matrix in so(3). *)
                (* Example Input: *)

                (* clear; clc; *)
                (* omg = [1; 2; 3]; *)
                (* so3mat = VecToso3(omg) *)

                (* Output: *)
                (* so3mat = *)
                (* 0    -3     2 *)
                (* 3     0    -1 *)
                (* -2     1     0 *)
                (* 'VecToso3:17' so3mat = [0, -omg(3), omg(2); omg(3), 0, -omg(1); -omg(2), omg(1), 0]; *)
                tmp_3[3] :=  -a_0[14];
                tmp_3[6] := a_0[13];
                tmp_3[1] := a_0[14];
                tmp_3[7] :=  -a_0[12];
                tmp_3[2] :=  -a_0[13];
                tmp_3[5] := a_0[12];
                FOR i_0 := 0 TO 2 DO
                    x_tmp := tmp_3[i_0 + 3];
                    thetalist0_0 := tmp_3[i_0];
                    g_a := tmp_3[i_0 + 6];
                    FOR omgmat_tmp := 0 TO 2 DO
                        R_tmp := DWORD_TO_DINT(SHL(DINT_TO_DWORD(omgmat_tmp), 2));
                        tmp_0[i_0 + (3 * omgmat_tmp)] := ((a_0[R_tmp + 1] * x_tmp) + (a_0[R_tmp] * thetalist0_0)) + (a_0[R_tmp + 2] * g_a);
                        Tsb_0[omgmat_tmp + (6 * i_0)] := a_0[(i_0 * 4) + omgmat_tmp];
                        Tsb_0[omgmat_tmp + (6 * (i_0 + 3))] := 0.0;
                    END_FOR;
                END_FOR;
                FOR i_0 := 0 TO 2 DO
                    Tsb_0[(6 * i_0) + 3] := tmp_0[3 * i_0];
                    R_tmp := DWORD_TO_DINT(SHL(DINT_TO_DWORD(i_0), 2));
                    omgmat_tmp := 6 * (i_0 + 3);
                    Tsb_0[omgmat_tmp + 3] := a_0[R_tmp];
                    Tsb_0[(6 * i_0) + 4] := tmp_0[(3 * i_0) + 1];
                    Tsb_0[omgmat_tmp + 4] := a_0[R_tmp + 1];
                    Tsb_0[(6 * i_0) + 5] := tmp_0[(3 * i_0) + 2];
                    Tsb_0[omgmat_tmp + 5] := a_0[R_tmp + 2];
                END_FOR;
                FOR i_0 := 0 TO 5 DO
                    thetalist0_0 := 0.0;
                    FOR omgmat_tmp := 0 TO 5 DO
                        thetalist0_0 := (Constant5_Value[((d_i + 1) * 6) + omgmat_tmp] * Tsb_0[(6 * omgmat_tmp) + i_0]) + thetalist0_0;
                    END_FOR;
                    Js[i_0 + (6 * (d_i + 1))] := thetalist0_0;
                END_FOR;
            END_FOR;
            i0_pinv(A := Js);
            tmp_1 := i0_pinv.X;
            FOR i_0 := 0 TO 4 DO
                x_tmp := 0.0;
                FOR omgmat_tmp := 0 TO 5 DO
                    x_tmp := (tmp_1[(5 * omgmat_tmp) + i_0] * Vs[omgmat_tmp]) + x_tmp;
                END_FOR;
                thetalist0[i_0] := thetalist0[i_0] + x_tmp;
            END_FOR;
            (* 'IKinSpace:56' i = i + 1; *)
            i := i + 1;
            (* 'IKinSpace:57' Tsb = FKinSpace(M, Slist, thetalist); *)
            FOR i_0 := 0 TO 15 DO
                Tsb[i_0] := Constant4_Value[i_0];
            END_FOR;
            (* *** CHAPTER 4: FORWARD KINEMATICS *** *)
            (* Takes M: the home configuration (position and orientation) of the  *)
            (* end-effector, *)
            (* Slist: The joint screw axes in the space frame when the manipulator *)
            (* is at the home position, *)
            (* thetalist: A list of joint coordinates. *)
            (* Returns T in SE(3) representing the end-effector frame, when the joints  *)
            (* are at the specified coordinates (i.t.o Space Frame). *)
            (* Example Inputs: *)

            (* clear; clc; *)
            (* M = [[-1, 0, 0, 0]; [0, 1, 0, 6]; [0, 0, -1, 2]; [0, 0, 0, 1]]; *)
            (* Slist = [[0; 0;  1;  4; 0;    0], ... *)
            (* [0; 0;  0;  0; 1;    0], ... *)
            (* [0; 0; -1; -6; 0; -0.1]]; *)
            (* thetalist =[pi / 2; 3; pi]; *)
            (* T = FKinSpace(M, Slist, thetalist) *)

            (* Output: *)
            (* T = *)
            (* -0.0000    1.0000         0   -5.0000 *)
            (* 1.0000    0.0000         0    4.0000 *)
            (* 0         0   -1.0000    1.6858 *)
            (* 0         0         0    1.0000 *)
            (* 'FKinSpace:27' T = M; *)
            (* 'FKinSpace:28' for i = size(thetalist, 1): -1: 1 *)
            se3mat[0] := 0.0;
            se3mat[5] := 0.0;
            se3mat[10] := 0.0;
            se3mat[3] := 0.0;
            se3mat[7] := 0.0;
            se3mat[11] := 0.0;
            se3mat[15] := 0.0;
            FOR e_i := 0 TO 4 DO
                (* 'FKinSpace:29' T = MatrixExp6(VecTose3(Slist(:, i) * thetalist(i))) * T; *)
                thetalist0_0 := thetalist0[4 - e_i];
                FOR i_0 := 0 TO 5 DO
                    V[i_0] := Constant5_Value[((4 - e_i) * 6) + i_0] * thetalist0_0;
                END_FOR;
                (* *** CHAPTER 3: RIGID-BODY MOTIONS *** *)
                (* Takes a 6-vector (representing a spatial velocity). *)
                (* Returns the corresponding 4x4 se(3) matrix. *)
                (* Example Input: *)

                (* clear; clc; *)
                (* V = [1; 2; 3; 4; 5; 6]; *)
                (* se3mat = VecTose3(V) *)

                (* Output: *)
                (* se3mat = *)
                (* 0    -3     2     4 *)
                (* 3     0    -1     5 *)
                (* -2     1     0     6 *)
                (* 0     0     0     0  *)
                (* 'VecTose3:18' se3mat = [VecToso3(V(1: 3)), V(4: 6); 0, 0, 0, 0]; *)
                (* *** CHAPTER 3: RIGID-BODY MOTIONS *** *)
                (* Takes a 3-vector (angular velocity). *)
                (* Returns the skew symmetric matrix in so(3). *)
                (* Example Input: *)

                (* clear; clc; *)
                (* omg = [1; 2; 3]; *)
                (* so3mat = VecToso3(omg) *)

                (* Output: *)
                (* so3mat = *)
                (* 0    -3     2 *)
                (* 3     0    -1 *)
                (* -2     1     0 *)
                (* 'VecToso3:17' so3mat = [0, -omg(3), omg(2); omg(3), 0, -omg(1); -omg(2), omg(1), 0]; *)
                se3mat[4] :=  -V[2];
                se3mat[8] := V[1];
                se3mat[1] := V[2];
                se3mat[9] :=  -V[0];
                se3mat[2] :=  -V[1];
                se3mat[6] := V[0];
                se3mat[12] := V[3];
                se3mat[13] := V[4];
                se3mat[14] := V[5];
                (* *** CHAPTER 3: RIGID-BODY MOTIONS *** *)
                (* Takes a se(3) representation of exponential coordinates. *)
                (* Returns a T matrix in SE(3) that is achieved by traveling along/about the  *)
                (* screw axis S for a distance theta from an initial configuration T = I. *)
                (* Example Input: *)

                (* clear; clc; *)
                (* se3mat = [ 0,      0,       0,      0; *)
                (* 0,      0, -1.5708, 2.3562; *)
                (* 0, 1.5708,       0, 2.3562; *)
                (* 0,      0,       0,      0] *)
                (* T = MatrixExp6(se3mat) *)

                (* Output: *)
                (* T = *)
                (* 1.0000         0         0         0 *)
                (* 0    0.0000   -1.0000   -0.0000 *)
                (* 0    1.0000    0.0000    3.0000 *)
                (* 0         0         0    1.0000  *)
                (* 'MatrixExp6:22' omgtheta = so3ToVec(se3mat(1: 3, 1: 3)); *)
                (* *** CHAPTER 3: RIGID-BODY MOTIONS *** *)
                (* Takes a 3x3 skew-symmetric matrix (an element of so(3)). *)
                (* Returns the corresponding 3-vector (angular velocity). *)
                (* Example Input:  *)

                (* clear; clc; *)
                (* so3mat = [[0, -3, 2]; [3, 0, -1]; [-2, 1, 0]]; *)
                (* omg = so3ToVec(so3mat)   *)

                (* Output: *)
                (* omg = *)
                (* 1 *)
                (* 2 *)
                (* 3 *)
                (* 'so3ToVec:17' omg = [so3mat(3, 2); so3mat(1, 3); so3mat(2, 1)]; *)
                omgtheta[0] := V[0];
                omgtheta[1] := V[1];
                omgtheta[2] := V[2];
                (* 'MatrixExp6:23' if NearZero(norm(omgtheta)) *)
                (* *** BASIC HELPER FUNCTIONS *** *)
                (* Takes a scalar. *)
                (* Checks if the scalar is small enough to be neglected. *)
                (* Example Input: *)

                (* clear; clc; *)
                (* near = -1e-7; *)
                (* judge = NearZero(near) *)

                (* Output: *)
                (* judge = *)
                (* 1 *)
                (* 'NearZero:15' judge = norm(near) < 1e-6; *)
                f_theta := norm(x := omgtheta);
                IF ABS(f_theta) < 1.0E-6 THEN
                    (* 'MatrixExp6:24' T = [eye(3), se3mat(1: 3, 4); 0, 0, 0, 1]; *)
                    i0_eye();
                    tmp_0 := i0_eye.I;
                    FOR i_0 := 0 TO 2 DO
                        R_tmp := DWORD_TO_DINT(SHL(DINT_TO_DWORD(i_0), 2));
                        a[R_tmp] := tmp_0[3 * i_0];
                        a[R_tmp + 1] := tmp_0[(3 * i_0) + 1];
                        a[R_tmp + 2] := tmp_0[(3 * i_0) + 2];
                        a[i_0 + 12] := se3mat[i_0 + 12];
                    END_FOR;
                    a[3] := 0.0;
                    a[7] := 0.0;
                    a[11] := 0.0;
                    a[15] := 1.0;
                ELSE
                    (* 'MatrixExp6:25' else *)
                    (* 'MatrixExp6:26' [omghat, theta] = AxisAng3(omgtheta); *)
                    (* *** CHAPTER 3: RIGID-BODY MOTIONS *** *)
                    (* Takes A 3-vector of exponential coordinates for rotation. *)
                    (* Returns the unit rotation axis omghat and the corresponding rotation  *)
                    (* angle theta. *)
                    (* Example Input: *)

                    (* clear; clc; *)
                    (* expc3 = [1; 2; 3]; *)
                    (* [omghat, theta] = AxisAng3(expc3)   *)

                    (* Output: *)
                    (* omghat = *)
                    (* 0.2673 *)
                    (* 0.5345 *)
                    (* 0.8018 *)
                    (* theta = *)
                    (* 3.7417 *)
                    (* 'AxisAng3:20' theta = norm(expc3); *)
                    (* 'AxisAng3:21' omghat = expc3 / theta; *)
                    (* 'MatrixExp6:27' omgmat = se3mat(1: 3, 1: 3) / theta; *)
                    FOR i_0 := 0 TO 2 DO
                        omgmat_tmp := DWORD_TO_DINT(SHL(DINT_TO_DWORD(i_0), 2));
                        omgmat[3 * i_0] := se3mat[omgmat_tmp] / f_theta;
                        omgmat[(3 * i_0) + 1] := se3mat[omgmat_tmp + 1] / f_theta;
                        omgmat[(3 * i_0) + 2] := se3mat[omgmat_tmp + 2] / f_theta;
                    END_FOR;
                    (* 'MatrixExp6:28' T = [MatrixExp3(se3mat(1: 3, 1: 3)), ... *)
                    (* 'MatrixExp6:29'          (eye(3) * theta + (1 - cos(theta)) * omgmat ... *)
                    (* 'MatrixExp6:30'           + (theta - sin(theta)) * omgmat * omgmat) ... *)
                    (* 'MatrixExp6:31'             * se3mat(1: 3, 4) / theta; *)
                    (* 'MatrixExp6:32'          0, 0, 0, 1]; *)
                    thetalist0_0 := 1.0 - COS(f_theta);
                    g_a := f_theta - SIN(f_theta);
                    (* *** CHAPTER 3: RIGID-BODY MOTIONS *** *)
                    (* Takes a 3x3 so(3) representation of exponential coordinates. *)
                    (* Returns R in SO(3) that is achieved by rotating about omghat by theta  *)
                    (* from an initial orientation R = I. *)
                    (* Example Input: *)

                    (* clear; clc; *)
                    (* so3mat = [[0, -3, 2]; [3, 0, -1]; [-2, 1, 0]]; *)
                    (* R = MatrixExp3(so3mat)   *)

                    (* Output: *)
                    (* R = *)
                    (* -0.6949    0.7135    0.0893 *)
                    (* -0.1920   -0.3038    0.9332 *)
                    (* 0.6930    0.6313    0.3481 *)
                    (* 'MatrixExp3:18' omgtheta = so3ToVec(so3mat); *)
                    (* *** CHAPTER 3: RIGID-BODY MOTIONS *** *)
                    (* Takes a 3x3 skew-symmetric matrix (an element of so(3)). *)
                    (* Returns the corresponding 3-vector (angular velocity). *)
                    (* Example Input:  *)

                    (* clear; clc; *)
                    (* so3mat = [[0, -3, 2]; [3, 0, -1]; [-2, 1, 0]]; *)
                    (* omg = so3ToVec(so3mat)   *)

                    (* Output: *)
                    (* omg = *)
                    (* 1 *)
                    (* 2 *)
                    (* 3 *)
                    (* 'so3ToVec:17' omg = [so3mat(3, 2); so3mat(1, 3); so3mat(2, 1)]; *)
                    omgtheta[0] := V[0];
                    omgtheta[1] := V[1];
                    omgtheta[2] := V[2];
                    (* 'MatrixExp3:19' if NearZero(norm(omgtheta)) *)
                    (* *** BASIC HELPER FUNCTIONS *** *)
                    (* Takes a scalar. *)
                    (* Checks if the scalar is small enough to be neglected. *)
                    (* Example Input: *)

                    (* clear; clc; *)
                    (* near = -1e-7; *)
                    (* judge = NearZero(near) *)

                    (* Output: *)
                    (* judge = *)
                    (* 1 *)
                    (* 'NearZero:15' judge = norm(near) < 1e-6; *)
                    j_theta := norm(x := omgtheta);
                    IF ABS(j_theta) < 1.0E-6 THEN
                        (* 'MatrixExp3:20' R = eye(3); *)
                        i0_eye();
                        b_R := i0_eye.I;
                    ELSE
                        (* 'MatrixExp3:21' else *)
                        (* 'MatrixExp3:22' [omghat, theta] = AxisAng3(omgtheta); *)
                        (* *** CHAPTER 3: RIGID-BODY MOTIONS *** *)
                        (* Takes A 3-vector of exponential coordinates for rotation. *)
                        (* Returns the unit rotation axis omghat and the corresponding rotation  *)
                        (* angle theta. *)
                        (* Example Input: *)

                        (* clear; clc; *)
                        (* expc3 = [1; 2; 3]; *)
                        (* [omghat, theta] = AxisAng3(expc3)   *)

                        (* Output: *)
                        (* omghat = *)
                        (* 0.2673 *)
                        (* 0.5345 *)
                        (* 0.8018 *)
                        (* theta = *)
                        (* 3.7417 *)
                        (* 'AxisAng3:20' theta = norm(expc3); *)
                        (* 'AxisAng3:21' omghat = expc3 / theta; *)
                        (* 'MatrixExp3:23' omgmat = so3mat / theta; *)
                        FOR i_0 := 0 TO 2 DO
                            omgmat_tmp := DWORD_TO_DINT(SHL(DINT_TO_DWORD(i_0), 2));
                            b_omgmat[3 * i_0] := se3mat[omgmat_tmp] / j_theta;
                            b_omgmat[(3 * i_0) + 1] := se3mat[omgmat_tmp + 1] / j_theta;
                            b_omgmat[(3 * i_0) + 2] := se3mat[omgmat_tmp + 2] / j_theta;
                        END_FOR;
                        (* 'MatrixExp3:24' R = eye(3) + sin(theta) * omgmat + (1 - cos(theta)) * omgmat * omgmat; *)
                        l_a := SIN(j_theta);
                        x_tmp := COS(j_theta);
                        i0_eye();
                        tmp_0 := i0_eye.I;
                        FOR i_0 := 0 TO 2 DO
                            FOR omgmat_tmp := 0 TO 2 DO
                                R_tmp := (3 * omgmat_tmp) + i_0;
                                b_R[R_tmp] := (((((1.0 - x_tmp) * b_omgmat[i_0 + 3]) * b_omgmat[(3 * omgmat_tmp) + 1]) + (((1.0 - x_tmp) * b_omgmat[i_0]) * b_omgmat[3 * omgmat_tmp])) + ((b_omgmat[i_0 + 6] * (1.0 - x_tmp)) * b_omgmat[(3 * omgmat_tmp) + 2])) + ((b_omgmat[R_tmp] * l_a) + tmp_0[R_tmp]);
                            END_FOR;
                        END_FOR;
                    END_IF;
                    FOR i_0 := 0 TO 2 DO
                        x_tmp := 0.0;
                        FOR omgmat_tmp := 0 TO 2 DO
                            R_tmp := (3 * omgmat_tmp) + i_0;
                            x_tmp := ((((((omgmat[i_0 + 3] * g_a) * omgmat[(3 * omgmat_tmp) + 1]) + ((g_a * omgmat[i_0]) * omgmat[3 * omgmat_tmp])) + ((omgmat[i_0 + 6] * g_a) * omgmat[(3 * omgmat_tmp) + 2])) + ((SINT_TO_LREAL(p_a[R_tmp]) * f_theta) + (omgmat[R_tmp] * thetalist0_0))) * se3mat[omgmat_tmp + 12]) + x_tmp;
                            a[omgmat_tmp + (i_0 * 4)] := b_R[(3 * i_0) + omgmat_tmp];
                        END_FOR;
                        a[i_0 + 12] := x_tmp / f_theta;
                    END_FOR;
                    a[3] := 0.0;
                    a[7] := 0.0;
                    a[11] := 0.0;
                    a[15] := 1.0;
                END_IF;
                FOR i_0 := 0 TO 3 DO
                    thetalist0_0 := a[i_0 + 4];
                    g_a := a[i_0];
                    l_a := a[i_0 + 8];
                    x_tmp := a[i_0 + 12];
                    FOR omgmat_tmp := 0 TO 3 DO
                        R_tmp := DWORD_TO_DINT(SHL(DINT_TO_DWORD(omgmat_tmp), 2));
                        a_0[i_0 + R_tmp] := (((Tsb[R_tmp + 1] * thetalist0_0) + (Tsb[R_tmp] * g_a)) + (Tsb[R_tmp + 2] * l_a)) + (Tsb[R_tmp + 3] * x_tmp);
                    END_FOR;
                END_FOR;
                FOR i_0 := 0 TO 15 DO
                    Tsb[i_0] := a_0[i_0];
                END_FOR;
            END_FOR;
            (* 'IKinSpace:58' Vs = Adjoint(Tsb) * se3ToVec(MatrixLog6(TransInv(Tsb) * T)); *)
            (* *** CHAPTER 3: RIGID-BODY MOTIONS *** *)
            (* Takes a transformation matrix T. *)
            (* Returns its inverse.  *)
            (* Uses the structure of transformation matrices to avoid taking a matrix *)
            (* inverse, for efficiency. *)
            (* Example Input: *)

            (* clear; clc; *)
            (* T = [[1, 0, 0, 0]; [0, 0, -1, 0]; [0, 1, 0, 3]; [0, 0, 0, 1]]; *)
            (* invT = TransInv(T) *)

            (* Ouput: *)
            (* invT = *)
            (* 1     0     0     0 *)
            (* 0     0     1    -3 *)
            (* 0    -1     0     0 *)
            (* 0     0     0     1 *)
            (* 'TransInv:20' [R, p] = TransToRp(T); *)
            (* *** CHAPTER 3: RIGID-BODY MOTIONS *** *)
            (* Takes the transformation matrix T in SE(3)  *)
            (* Returns R: the corresponding rotation matrix *)
            (* p: the corresponding position vector . *)
            (* Example Input: *)

            (* clear; clc; *)
            (* T = [[1, 0, 0, 0]; [0, 0, -1, 0]; [0, 1, 0, 3]; [0, 0, 0, 1]]; *)
            (* [R, p] = TransToRp(T) *)

            (* Output: *)
            (* R = *)
            (* 1     0     0 *)
            (* 0     0    -1 *)
            (* 0     1     0 *)
            (* p = *)
            (* 0 *)
            (* 0 *)
            (* 3 *)
            (* 'TransToRp:22' R = T(1: 3, 1: 3); *)
            (* 'TransToRp:23' p = T(1: 3, 4); *)
            (* 'TransInv:21' invT = [transpose(R), -transpose(R) * p; 0, 0, 0, 1]; *)
            FOR i_0 := 0 TO 2 DO
                omgmat[3 * i_0] := Tsb[i_0];
                omgmat[(3 * i_0) + 1] := Tsb[i_0 + 4];
                omgmat[(3 * i_0) + 2] := Tsb[i_0 + 8];
            END_FOR;
            FOR i_0 := 0 TO 8 DO
                b_R[i_0] :=  -omgmat[i_0];
            END_FOR;
            thetalist0_0 := Tsb[13];
            g_a := Tsb[12];
            l_a := Tsb[14];
            FOR i_0 := 0 TO 2 DO
                omgmat_tmp := DWORD_TO_DINT(SHL(DINT_TO_DWORD(i_0), 2));
                se3mat[omgmat_tmp] := omgmat[3 * i_0];
                se3mat[omgmat_tmp + 1] := omgmat[(3 * i_0) + 1];
                se3mat[omgmat_tmp + 2] := omgmat[(3 * i_0) + 2];
                se3mat[i_0 + 12] := ((b_R[i_0 + 3] * thetalist0_0) + (b_R[i_0] * g_a)) + (b_R[i_0 + 6] * l_a);
            END_FOR;
            se3mat[3] := 0.0;
            se3mat[7] := 0.0;
            se3mat[11] := 0.0;
            se3mat[15] := 1.0;
            FOR i_0 := 0 TO 3 DO
                thetalist0_0 := se3mat[i_0 + 4];
                g_a := se3mat[i_0];
                l_a := se3mat[i_0 + 8];
                x_tmp := se3mat[i_0 + 12];
                FOR omgmat_tmp := 0 TO 3 DO
                    R_tmp := DWORD_TO_DINT(SHL(DINT_TO_DWORD(omgmat_tmp), 2));
                    a_0[i_0 + R_tmp] := (((T[R_tmp + 1] * thetalist0_0) + (T[R_tmp] * g_a)) + (T[R_tmp + 2] * l_a)) + (T[R_tmp + 3] * x_tmp);
                END_FOR;
            END_FOR;
            (* *** CHAPTER 3: RIGID-BODY MOTIONS *** *)
            (* Takes a transformation matrix T in SE(3). *)
            (* Returns the corresponding se(3) representation of exponential  *)
            (* coordinates. *)
            (* Example Input: *)

            (* clear; clc; *)
            (* T = [[1, 0, 0, 0]; [0, 0, -1, 0]; [0, 1, 0, 3]; [0, 0, 0, 1]]; *)
            (* expmat = MatrixLog6(T) *)

            (* Output: *)
            (* expc6 = *)
            (* 0         0         0         0 *)
            (* 0         0   -1.5708    2.3562 *)
            (* 0    1.5708         0    2.3562 *)
            (* 0         0         0         0 *)
            (* 'MatrixLog6:19' [R, p] = TransToRp(T); *)
            (* *** CHAPTER 3: RIGID-BODY MOTIONS *** *)
            (* Takes the transformation matrix T in SE(3)  *)
            (* Returns R: the corresponding rotation matrix *)
            (* p: the corresponding position vector . *)
            (* Example Input: *)

            (* clear; clc; *)
            (* T = [[1, 0, 0, 0]; [0, 0, -1, 0]; [0, 1, 0, 3]; [0, 0, 0, 1]]; *)
            (* [R, p] = TransToRp(T) *)

            (* Output: *)
            (* R = *)
            (* 1     0     0 *)
            (* 0     0    -1 *)
            (* 0     1     0 *)
            (* p = *)
            (* 0 *)
            (* 0 *)
            (* 3 *)
            (* 'TransToRp:22' R = T(1: 3, 1: 3); *)
            (* 'TransToRp:23' p = T(1: 3, 4); *)
            (* 'MatrixLog6:20' omgmat = MatrixLog3(R); *)
            FOR i_0 := 0 TO 2 DO
                R_tmp := DWORD_TO_DINT(SHL(DINT_TO_DWORD(i_0), 2));
                b_R[3 * i_0] := a_0[R_tmp];
                b_R[(3 * i_0) + 1] := a_0[R_tmp + 1];
                b_R[(3 * i_0) + 2] := a_0[R_tmp + 2];
            END_FOR;
            i0_MatrixLog3(b_R := b_R);
            omgmat := i0_MatrixLog3.so3mat;
            (* 'MatrixLog6:21' if isequal(omgmat, zeros(3)) *)
            IF isequal(varargin_1 := omgmat, varargin_2 := tmp_2) THEN
                (* 'MatrixLog6:22' expmat = [zeros(3), T(1: 3, 4); 0, 0, 0, 0]; *)
                FOR i_0 := 0 TO 2 DO
                    omgmat_tmp := DWORD_TO_DINT(SHL(DINT_TO_DWORD(i_0), 2));
                    se3mat[omgmat_tmp] := 0.0;
                    se3mat[omgmat_tmp + 1] := 0.0;
                    se3mat[omgmat_tmp + 2] := 0.0;
                    se3mat[i_0 + 12] := a_0[i_0 + 12];
                END_FOR;
                se3mat[3] := 0.0;
                se3mat[7] := 0.0;
                se3mat[11] := 0.0;
                se3mat[15] := 0.0;
            ELSE
                (* 'MatrixLog6:23' else *)
                (* 'MatrixLog6:24' theta = acos((trace(R) - 1) / 2); *)
                b_theta := ACOS((((a_0[0] + a_0[5]) + a_0[10]) - 1.0) / 2.0);
                (* 'MatrixLog6:25' expmat = [omgmat, (eye(3) - omgmat / 2 ... *)
                (* 'MatrixLog6:26'                       + (1 / theta - cot(theta / 2) / 2) ... *)
                (* 'MatrixLog6:27'                         * omgmat * omgmat / theta) * p; *)
                (* 'MatrixLog6:28'               0, 0, 0, 0]; *)
                thetalist0_0 := (1.0 / b_theta) - ((1.0 / TAN(b_theta / 2.0)) / 2.0);
                i0_eye();
                tmp_0 := i0_eye.I;
                FOR i_0 := 0 TO 2 DO
                    x_tmp := 0.0;
                    FOR omgmat_tmp := 0 TO 2 DO
                        R_tmp := (3 * omgmat_tmp) + i_0;
                        x_tmp := (((((((omgmat[i_0 + 3] * thetalist0_0) * omgmat[(3 * omgmat_tmp) + 1]) + ((thetalist0_0 * omgmat[i_0]) * omgmat[3 * omgmat_tmp])) + ((omgmat[i_0 + 6] * thetalist0_0) * omgmat[(3 * omgmat_tmp) + 2])) / b_theta) + (tmp_0[R_tmp] - (omgmat[R_tmp] / 2.0))) * a_0[omgmat_tmp + 12]) + x_tmp;
                        se3mat[omgmat_tmp + (i_0 * 4)] := omgmat[(3 * i_0) + omgmat_tmp];
                    END_FOR;
                    se3mat[i_0 + 12] := x_tmp;
                END_FOR;
                se3mat[3] := 0.0;
                se3mat[7] := 0.0;
                se3mat[11] := 0.0;
                se3mat[15] := 0.0;
            END_IF;
            (* *** CHAPTER 3: RIGID-BODY MOTIONS *** *)
            (* Takes T a transformation matrix SE3.  *)
            (* Returns the corresponding 6x6 adjoint representation [AdT]. *)
            (* Example Input: *)

            (* clear; clc; *)
            (* T = [[1, 0, 0, 0]; [0, 0, -1, 0]; [0, 1, 0, 3]; [0, 0, 0, 1]]; *)
            (* AdT = Adjoint(T) *)

            (* Output: *)
            (* AdT = *)
            (* 1     0     0     0     0     0 *)
            (* 0     0    -1     0     0     0 *)
            (* 0     1     0     0     0     0 *)
            (* 0     0     3     1     0     0 *)
            (* 3     0     0     0     0    -1 *)
            (* 0     0     0     0     1     0 *)
            (* 'Adjoint:20' [R, p] = TransToRp(T); *)
            (* *** CHAPTER 3: RIGID-BODY MOTIONS *** *)
            (* Takes the transformation matrix T in SE(3)  *)
            (* Returns R: the corresponding rotation matrix *)
            (* p: the corresponding position vector . *)
            (* Example Input: *)

            (* clear; clc; *)
            (* T = [[1, 0, 0, 0]; [0, 0, -1, 0]; [0, 1, 0, 3]; [0, 0, 0, 1]]; *)
            (* [R, p] = TransToRp(T) *)

            (* Output: *)
            (* R = *)
            (* 1     0     0 *)
            (* 0     0    -1 *)
            (* 0     1     0 *)
            (* p = *)
            (* 0 *)
            (* 0 *)
            (* 3 *)
            (* 'TransToRp:22' R = T(1: 3, 1: 3); *)
            (* 'TransToRp:23' p = T(1: 3, 4); *)
            (* 'Adjoint:21' AdT = [R, zeros(3); VecToso3(p) * R, R]; *)
            (* *** CHAPTER 3: RIGID-BODY MOTIONS *** *)
            (* Takes a 3-vector (angular velocity). *)
            (* Returns the skew symmetric matrix in so(3). *)
            (* Example Input: *)

            (* clear; clc; *)
            (* omg = [1; 2; 3]; *)
            (* so3mat = VecToso3(omg) *)

            (* Output: *)
            (* so3mat = *)
            (* 0    -3     2 *)
            (* 3     0    -1 *)
            (* -2     1     0 *)
            (* 'VecToso3:17' so3mat = [0, -omg(3), omg(2); omg(3), 0, -omg(1); -omg(2), omg(1), 0]; *)
            (* *** CHAPTER 3: RIGID-BODY MOTIONS *** *)
            (* Takes se3mat a 4x4 se(3) matrix *)
            (* Returns the corresponding 6-vector (representing spatial velocity). *)
            (* Example Input: *)

            (* clear; clc; *)
            (* se3mat = [[0, -3, 2, 4]; [3, 0, -1, 5]; [-2, 1, 0, 6]; [0, 0, 0, 0]]; *)
            (* V = se3ToVec(se3mat) *)

            (* Output: *)
            (* V = *)
            (* 1 *)
            (* 2 *)
            (* 3 *)
            (* 4 *)
            (* 5 *)
            (* 6 *)
            (* 'se3ToVec:20' V = [se3mat(3, 2); se3mat(1, 3); se3mat(2, 1); se3mat(1: 3, 4)]; *)
            tmp_4[3] :=  -Tsb[14];
            tmp_4[6] := Tsb[13];
            tmp_4[1] := Tsb[14];
            tmp_4[7] :=  -Tsb[12];
            tmp_4[2] :=  -Tsb[13];
            tmp_4[5] := Tsb[12];
            FOR i_0 := 0 TO 2 DO
                x_tmp := tmp_4[i_0 + 3];
                thetalist0_0 := tmp_4[i_0];
                g_a := tmp_4[i_0 + 6];
                FOR omgmat_tmp := 0 TO 2 DO
                    R_tmp := DWORD_TO_DINT(SHL(DINT_TO_DWORD(omgmat_tmp), 2));
                    tmp_0[i_0 + (3 * omgmat_tmp)] := ((Tsb[R_tmp + 1] * x_tmp) + (Tsb[R_tmp] * thetalist0_0)) + (Tsb[R_tmp + 2] * g_a);
                    Tsb_0[omgmat_tmp + (6 * i_0)] := Tsb[(i_0 * 4) + omgmat_tmp];
                    Tsb_0[omgmat_tmp + (6 * (i_0 + 3))] := 0.0;
                END_FOR;
            END_FOR;
            V[0] := se3mat[6];
            V[1] := se3mat[8];
            V[2] := se3mat[1];
            FOR i_0 := 0 TO 2 DO
                Tsb_0[(6 * i_0) + 3] := tmp_0[3 * i_0];
                omgmat_tmp := DWORD_TO_DINT(SHL(DINT_TO_DWORD(i_0), 2));
                R_tmp := 6 * (i_0 + 3);
                Tsb_0[R_tmp + 3] := Tsb[omgmat_tmp];
                Tsb_0[(6 * i_0) + 4] := tmp_0[(3 * i_0) + 1];
                Tsb_0[R_tmp + 4] := Tsb[omgmat_tmp + 1];
                Tsb_0[(6 * i_0) + 5] := tmp_0[(3 * i_0) + 2];
                Tsb_0[R_tmp + 5] := Tsb[omgmat_tmp + 2];
                V[i_0 + 3] := se3mat[i_0 + 12];
            END_FOR;
            FOR i_0 := 0 TO 5 DO
                thetalist0_0 := 0.0;
                FOR omgmat_tmp := 0 TO 5 DO
                    thetalist0_0 := (Tsb_0[(6 * omgmat_tmp) + i_0] * V[omgmat_tmp]) + thetalist0_0;
                END_FOR;
                Vs[i_0] := thetalist0_0;
            END_FOR;
            (* 'IKinSpace:59' err = norm(Vs(1: 3)) > eomg || norm(Vs(4: 6)) > ev; *)
            se3mat_0[0] := Vs[0];
            se3mat_0[1] := Vs[1];
            se3mat_0[2] := Vs[2];
            IF norm(x := se3mat_0) <= 1.0E-5 THEN
                se3mat_0[0] := Vs[3];
                se3mat_0[1] := Vs[4];
                se3mat_0[2] := Vs[5];
                IF norm(x := se3mat_0) <= 1.0E-7 THEN
                    err := FALSE;
                END_IF;
            END_IF;
        END_WHILE;
        (* End of Outputs for SubSystem: '<Root>/FB_InverceKinematics' *)
        (* 'IKinSpace:61' success = ~ err; *)
        (* Assign them to the pre-allocated outputs *)
        (* '<S2>:1:23' thetaList    = thetaOut; *)
        (* '<S2>:1:24' success      = successOut; *)
        (* '<S2>:1:27' Js = JacobianSpace(SList,thetaList); *)
        (* *** CHAPTER 5: VELOCITY KINEMATICS AND STATICS *** *)
        (* Takes Slist: The joint screw axes in the space frame when the manipulator *)
        (* is at the home position, in the format of a matrix with the *)
        (* screw axes as the columns, *)
        (* thetalist: A list of joint coordinates.  *)
        (* Returns the corresponding space Jacobian (6xn real numbers). *)
        (* Example Input: *)

        (* clear; clc; *)
        (* Slist = [[0; 0; 1;   0; 0.2; 0.2], ... *)
        (* [1; 0; 0;   2;   0;   3], ... *)
        (* [0; 1; 0;   0;   2;   1], ... *)
        (* [1; 0; 0; 0.2; 0.3; 0.4]]; *)
        (* thetalist = [0.2; 1.1; 0.1; 1.2]; *)
        (* Js = JacobianSpace(Slist, thetalist) *)

        (* Output: *)
        (* Js = *)
        (* 0    0.9801   -0.0901    0.9575 *)
        (* 0    0.1987    0.4446    0.2849 *)
        (* 1.0000         0    0.8912   -0.0453 *)
        (* 0    1.9522   -2.2164   -0.5116 *)
        (* 0.2000    0.4365   -2.4371    2.7754 *)
        (* 0.2000    2.9603    3.2357    2.2251 *)
        (* 'JacobianSpace:27' Js = Slist; *)
        (* Outputs for Atomic SubSystem: '<Root>/FB_InverceKinematics' *)
        (* MATLAB Function: '<S1>/inverceKinematics' incorporates:
         *  Constant: '<S1>/Constant5' *)
        FOR i_0 := 0 TO 29 DO
            Js[i_0] := Constant5_Value[i_0];
        END_FOR;
        (* End of Outputs for SubSystem: '<Root>/FB_InverceKinematics' *)
        (* 'JacobianSpace:28' T = eye(4); *)
        (* Outputs for Atomic SubSystem: '<Root>/FB_InverceKinematics' *)
        (* MATLAB Function: '<S1>/inverceKinematics' *)
        FOR i_0 := 0 TO 15 DO
            T[i_0] := 0.0;
        END_FOR;
        T[0] := 1.0;
        T[5] := 1.0;
        T[10] := 1.0;
        T[15] := 1.0;
        (* End of Outputs for SubSystem: '<Root>/FB_InverceKinematics' *)
        (* 'JacobianSpace:29' for i = 2: length(thetalist) *)
        (* Outputs for Atomic SubSystem: '<Root>/FB_InverceKinematics' *)
        (* MATLAB Function: '<S1>/inverceKinematics' *)
        se3mat[0] := 0.0;
        se3mat[5] := 0.0;
        se3mat[10] := 0.0;
        se3mat[3] := 0.0;
        se3mat[7] := 0.0;
        se3mat[11] := 0.0;
        se3mat[15] := 0.0;
        (* End of Outputs for SubSystem: '<Root>/FB_InverceKinematics' *)
        (* Outputs for Atomic SubSystem: '<Root>/FB_InverceKinematics' *)
        (* MATLAB Function: '<S1>/inverceKinematics' *)
        tmp_0[0] := 0.0;
        tmp_0[4] := 0.0;
        tmp_0[8] := 0.0;
        (* End of Outputs for SubSystem: '<Root>/FB_InverceKinematics' *)
        (* Outputs for Atomic SubSystem: '<Root>/FB_InverceKinematics' *)
        (* MATLAB Function: '<S1>/inverceKinematics' incorporates:
         *  Constant: '<S1>/Constant5' *)
        FOR b_i := 0 TO 3 DO
            (* 'JacobianSpace:30' T = T * MatrixExp6(VecTose3(Slist(:, i - 1) * thetalist(i - 1))); *)
            thetalist0_0 := thetalist0[b_i];
            FOR i_0 := 0 TO 5 DO
                V[i_0] := Constant5_Value[(6 * b_i) + i_0] * thetalist0_0;
            END_FOR;
            (* *** CHAPTER 3: RIGID-BODY MOTIONS *** *)
            (* Takes a 6-vector (representing a spatial velocity). *)
            (* Returns the corresponding 4x4 se(3) matrix. *)
            (* Example Input: *)

            (* clear; clc; *)
            (* V = [1; 2; 3; 4; 5; 6]; *)
            (* se3mat = VecTose3(V) *)

            (* Output: *)
            (* se3mat = *)
            (* 0    -3     2     4 *)
            (* 3     0    -1     5 *)
            (* -2     1     0     6 *)
            (* 0     0     0     0  *)
            (* 'VecTose3:18' se3mat = [VecToso3(V(1: 3)), V(4: 6); 0, 0, 0, 0]; *)
            (* *** CHAPTER 3: RIGID-BODY MOTIONS *** *)
            (* Takes a 3-vector (angular velocity). *)
            (* Returns the skew symmetric matrix in so(3). *)
            (* Example Input: *)

            (* clear; clc; *)
            (* omg = [1; 2; 3]; *)
            (* so3mat = VecToso3(omg) *)

            (* Output: *)
            (* so3mat = *)
            (* 0    -3     2 *)
            (* 3     0    -1 *)
            (* -2     1     0 *)
            (* 'VecToso3:17' so3mat = [0, -omg(3), omg(2); omg(3), 0, -omg(1); -omg(2), omg(1), 0]; *)
            se3mat[4] :=  -V[2];
            se3mat[8] := V[1];
            se3mat[1] := V[2];
            se3mat[9] :=  -V[0];
            se3mat[2] :=  -V[1];
            se3mat[6] := V[0];
            se3mat[12] := V[3];
            se3mat[13] := V[4];
            se3mat[14] := V[5];
            (* *** CHAPTER 3: RIGID-BODY MOTIONS *** *)
            (* Takes a se(3) representation of exponential coordinates. *)
            (* Returns a T matrix in SE(3) that is achieved by traveling along/about the  *)
            (* screw axis S for a distance theta from an initial configuration T = I. *)
            (* Example Input: *)

            (* clear; clc; *)
            (* se3mat = [ 0,      0,       0,      0; *)
            (* 0,      0, -1.5708, 2.3562; *)
            (* 0, 1.5708,       0, 2.3562; *)
            (* 0,      0,       0,      0] *)
            (* T = MatrixExp6(se3mat) *)

            (* Output: *)
            (* T = *)
            (* 1.0000         0         0         0 *)
            (* 0    0.0000   -1.0000   -0.0000 *)
            (* 0    1.0000    0.0000    3.0000 *)
            (* 0         0         0    1.0000  *)
            (* 'MatrixExp6:22' omgtheta = so3ToVec(se3mat(1: 3, 1: 3)); *)
            (* *** CHAPTER 3: RIGID-BODY MOTIONS *** *)
            (* Takes a 3x3 skew-symmetric matrix (an element of so(3)). *)
            (* Returns the corresponding 3-vector (angular velocity). *)
            (* Example Input:  *)

            (* clear; clc; *)
            (* so3mat = [[0, -3, 2]; [3, 0, -1]; [-2, 1, 0]]; *)
            (* omg = so3ToVec(so3mat)   *)

            (* Output: *)
            (* omg = *)
            (* 1 *)
            (* 2 *)
            (* 3 *)
            (* 'so3ToVec:17' omg = [so3mat(3, 2); so3mat(1, 3); so3mat(2, 1)]; *)
            omgtheta[0] := V[0];
            omgtheta[1] := V[1];
            omgtheta[2] := V[2];
            (* 'MatrixExp6:23' if NearZero(norm(omgtheta)) *)
            (* *** BASIC HELPER FUNCTIONS *** *)
            (* Takes a scalar. *)
            (* Checks if the scalar is small enough to be neglected. *)
            (* Example Input: *)

            (* clear; clc; *)
            (* near = -1e-7; *)
            (* judge = NearZero(near) *)

            (* Output: *)
            (* judge = *)
            (* 1 *)
            (* 'NearZero:15' judge = norm(near) < 1e-6; *)
            c_theta := norm(x := omgtheta);
            IF ABS(c_theta) < 1.0E-6 THEN
                (* 'MatrixExp6:24' T = [eye(3), se3mat(1: 3, 4); 0, 0, 0, 1]; *)
                i0_eye();
                tmp := i0_eye.I;
                FOR i_0 := 0 TO 2 DO
                    R_tmp := DWORD_TO_DINT(SHL(DINT_TO_DWORD(i_0), 2));
                    a[R_tmp] := tmp[3 * i_0];
                    a[R_tmp + 1] := tmp[(3 * i_0) + 1];
                    a[R_tmp + 2] := tmp[(3 * i_0) + 2];
                    a[i_0 + 12] := se3mat[i_0 + 12];
                END_FOR;
                a[3] := 0.0;
                a[7] := 0.0;
                a[11] := 0.0;
                a[15] := 1.0;
            ELSE
                (* 'MatrixExp6:25' else *)
                (* 'MatrixExp6:26' [omghat, theta] = AxisAng3(omgtheta); *)
                (* *** CHAPTER 3: RIGID-BODY MOTIONS *** *)
                (* Takes A 3-vector of exponential coordinates for rotation. *)
                (* Returns the unit rotation axis omghat and the corresponding rotation  *)
                (* angle theta. *)
                (* Example Input: *)

                (* clear; clc; *)
                (* expc3 = [1; 2; 3]; *)
                (* [omghat, theta] = AxisAng3(expc3)   *)

                (* Output: *)
                (* omghat = *)
                (* 0.2673 *)
                (* 0.5345 *)
                (* 0.8018 *)
                (* theta = *)
                (* 3.7417 *)
                (* 'AxisAng3:20' theta = norm(expc3); *)
                (* 'AxisAng3:21' omghat = expc3 / theta; *)
                (* 'MatrixExp6:27' omgmat = se3mat(1: 3, 1: 3) / theta; *)
                FOR i_0 := 0 TO 2 DO
                    omgmat_tmp := DWORD_TO_DINT(SHL(DINT_TO_DWORD(i_0), 2));
                    omgmat[3 * i_0] := se3mat[omgmat_tmp] / c_theta;
                    omgmat[(3 * i_0) + 1] := se3mat[omgmat_tmp + 1] / c_theta;
                    omgmat[(3 * i_0) + 2] := se3mat[omgmat_tmp + 2] / c_theta;
                END_FOR;
                (* 'MatrixExp6:28' T = [MatrixExp3(se3mat(1: 3, 1: 3)), ... *)
                (* 'MatrixExp6:29'          (eye(3) * theta + (1 - cos(theta)) * omgmat ... *)
                (* 'MatrixExp6:30'           + (theta - sin(theta)) * omgmat * omgmat) ... *)
                (* 'MatrixExp6:31'             * se3mat(1: 3, 4) / theta; *)
                (* 'MatrixExp6:32'          0, 0, 0, 1]; *)
                thetalist0_0 := 1.0 - COS(c_theta);
                g_a := c_theta - SIN(c_theta);
                (* *** CHAPTER 3: RIGID-BODY MOTIONS *** *)
                (* Takes a 3x3 so(3) representation of exponential coordinates. *)
                (* Returns R in SO(3) that is achieved by rotating about omghat by theta  *)
                (* from an initial orientation R = I. *)
                (* Example Input: *)

                (* clear; clc; *)
                (* so3mat = [[0, -3, 2]; [3, 0, -1]; [-2, 1, 0]]; *)
                (* R = MatrixExp3(so3mat)   *)

                (* Output: *)
                (* R = *)
                (* -0.6949    0.7135    0.0893 *)
                (* -0.1920   -0.3038    0.9332 *)
                (* 0.6930    0.6313    0.3481 *)
                (* 'MatrixExp3:18' omgtheta = so3ToVec(so3mat); *)
                (* *** CHAPTER 3: RIGID-BODY MOTIONS *** *)
                (* Takes a 3x3 skew-symmetric matrix (an element of so(3)). *)
                (* Returns the corresponding 3-vector (angular velocity). *)
                (* Example Input:  *)

                (* clear; clc; *)
                (* so3mat = [[0, -3, 2]; [3, 0, -1]; [-2, 1, 0]]; *)
                (* omg = so3ToVec(so3mat)   *)
